SPLINE
SPL {X  -162.820, Y  +509.871, Z    +0.000, E1   +42.115, E3 +330842.346}
SPL {X  -162.820, Y  +501.934, Z    +0.000, E1   +43.022, E3 +330855.073}
SPL {X  -162.820, Y  +494.356, Z    +0.000, E1   +43.819, E3 +330866.915}
SPL {X  -162.820, Y  +487.058, Z    +0.000, E1   +44.544, E3 +330878.378}
SPL {X  -162.820, Y  +476.193, Z    +0.000, E1   +45.591, E3 +330894.817}
SPL {X  -162.820, Y  +465.836, Z    +0.000, E1   +46.727, E3 +330908.733}
SPL {X  -162.820, Y  +457.217, Z    +0.000, E1   +47.671, E3 +330919.772}
SPL {X  -162.820, Y  +446.677, Z    +0.000, E1   +48.707, E3 +330933.301}
SPL {X  -162.820, Y  +435.978, Z    +0.000, E1   +49.560, E3 +330947.450}
SPL {X  -162.820, Y  +428.488, Z    +0.000, E1   +49.830, E3 +330959.030}
SPL {X  -162.820, Y  +423.062, Z    +0.000, E1   +49.728, E3 +330969.173}
SPL {X  -162.820, Y  +416.560, Z    +0.000, E1   +49.816, E3 +330980.154}
SPL {X  -162.820, Y  +407.996, Z    +0.000, E1   +49.793, E3 +330995.519}
SPL {X  -162.820, Y  +398.766, Z    +0.000, E1   +49.793, E3 +331011.698}
SPL {X  -162.820, Y  +391.831, Z    +0.000, E1   +49.801, E3 +331023.744}
SPL {X  -162.820, Y  +386.334, Z    +0.000, E1   +49.739, E3 +331033.833}
SPL {X  -162.801, Y  +377.981, Z    +0.000, E1   +49.798, E3 +331048.354}
SPL {X  -162.314, Y  +367.677, Z    +0.000, E1   +49.734, E3 +331066.994}
SPL {X  -161.614, Y  +360.718, Z    +0.000, E1   +49.491, E3 +331080.412}
SPL {X  -160.828, Y  +355.106, Z    +0.000, E1   +49.536, E3 +331090.096}
SPL {X  -159.832, Y  +349.452, Z    +0.000, E1   +49.188, E3 +331102.067}
SPL {X  -158.863, Y  +344.823, Z    +0.000, E1   +49.020, E3 +331111.116}
SPL {X  -157.695, Y  +339.971, Z    +0.000, E1   +48.934, E3 +331120.212}
SPL {X  -156.136, Y  +334.326, Z    +0.000, E1   +48.578, E3 +331132.179}
SPL {X  -154.561, Y  +329.302, Z    +0.000, E1   +48.290, E3 +331142.509}
SPL {X  -152.787, Y  +324.229, Z    +0.000, E1   +47.981, E3 +331153.200}
SPL {X  -150.789, Y  +319.074, Z    +0.000, E1   +47.585, E3 +331164.222}
SPL {X  -145.123, Y  +306.679, Z    +0.000, E1   +50.518, E3 +331170.119}
SPL {X  -135.207, Y  +289.783, Z    +0.000, E1   +44.101, E3 +331263.634}
ENDSPLINE

SPLINE
SPL {X  -154.528, Y  +329.203, Z    +0.000, E1   +28.834, E3 +331333.995}
SPL {X  -160.380, Y  +352.419, Z    +0.000, E1   +18.163, E3 +331338.355}
SPL {X  -162.149, Y  +365.734, Z    +0.000, E1   +11.090, E3 +331336.964}
SPL {X  -162.754, Y  +375.862, Z    +0.000, E1    +5.134, E3 +331337.801}
SPL {X  -162.820, Y  +382.085, Z    +0.000, E1    +0.928, E3 +331337.489}
SPL {X  -162.820, Y  +385.149, Z    +0.000, E1    -1.602, E3 +331337.216}
SPL {X  -162.820, Y  +388.871, Z    +0.000, E1    -5.151, E3 +331337.171}
SPL {X  -162.820, Y  +395.861, Z    +0.000, E1   -13.028, E3 +331337.282}
SPL {X  -162.820, Y  +409.049, Z    +0.000, E1   -29.128, E3 +331336.125}
SPL {X  -162.820, Y  +446.299, Z    +0.000, E1   -49.360, E3 +331356.629}
SPL {X  -162.820, Y  +502.427, Z    +0.000, E1   -53.345, E3 +331419.614}
ENDSPLINE

SPLINE
SPL {X  -162.820, Y  +494.458, Z    +0.000, E1   -49.332, E3 +331430.146}
ENDSPLINE

SPLINE
SPL {X  -162.820, Y  +499.429, Z    +0.000, E1   -49.453, E3 +331438.355}
SPL {X  -162.820, Y  +505.173, Z    +0.000, E1   -49.386, E3 +331449.011}
SPL {X  -162.820, Y  +510.642, Z    +0.000, E1   -49.447, E3 +331458.361}
SPL {X  -162.820, Y  +516.435, Z    +0.000, E1   -49.526, E3 +331468.239}
SPL {X  -162.820, Y  +523.383, Z    +0.000, E1   -49.407, E3 +331481.426}
SPL {X  -162.820, Y  +530.598, Z    +0.000, E1   -49.471, E3 +331493.828}
SPL {X  -162.820, Y  +536.932, Z    +0.000, E1   -49.395, E3 +331505.585}
SPL {X  -162.820, Y  +543.021, Z    +0.000, E1   -49.432, E3 +331516.191}
SPL {X  -162.820, Y  +548.933, Z    +0.000, E1   -49.456, E3 +331526.595}
SPL {X  -162.820, Y  +553.997, Z    +0.000, E1   -49.325, E3 +331536.399}
SPL {X  -162.820, Y  +560.268, Z    +0.000, E1   -49.531, E3 +331546.357}
SPL {X  -162.820, Y  +564.590, Z    +0.000, E1   -49.361, E3 +331555.056}
SPL {X  -162.820, Y  +570.444, Z    +0.000, E1   -49.421, E3 +331565.208}
SPL {X  -162.820, Y  +577.429, Z    +0.000, E1   -49.474, E3 +331577.322}
SPL {X  -162.820, Y  +585.965, Z    +0.000, E1   -49.447, E3 +331592.896}
SPL {X  -162.820, Y  +594.192, Z    +0.000, E1   -49.325, E3 +331608.139}
SPL {X  -162.820, Y  +600.267, Z    +0.000, E1   -49.443, E3 +331618.228}
SPL {X  -162.820, Y  +606.218, Z    +0.000, E1   -49.464, E3 +331628.775}
SPL {X  -162.820, Y  +612.538, Z    +0.000, E1   -49.488, E3 +331639.826}
SPL {X  -162.820, Y  +617.738, Z    +0.000, E1   -49.301, E3 +331650.262}
SPL {X  -162.820, Y  +624.265, Z    +0.000, E1   -49.443, E3 +331661.057}
SPL {X  -162.820, Y  +632.551, Z    +0.000, E1   -49.478, E3 +331675.826}
SPL {X  -162.820, Y  +641.207, Z    +0.000, E1   -49.420, E3 +331691.469}
SPL {X  -162.820, Y  +649.864, Z    +0.000, E1   -49.433, E3 +331706.947}
SPL {X  -162.820, Y  +658.147, Z    +0.000, E1   -49.491, E3 +331721.214}
SPL {X  -162.820, Y  +663.916, Z    +0.000, E1   -49.371, E3 +331732.204}
SPL {X  -162.820, Y  +669.755, Z    +0.000, E1   -49.387, E3 +331742.529}
SPL {X  -162.807, Y  +675.597, Z    +0.000, E1   -49.472, E3 +331752.431}
SPL {X  -162.632, Y  +681.322, Z    +0.000, E1   -49.345, E3 +331763.443}
SPL {X  -162.228, Y  +687.372, Z    +0.000, E1   -49.294, E3 +331774.529}
SPL {X  -161.723, Y  +692.372, Z    +0.000, E1   -49.172, E3 +331784.159}
SPL {X  -161.009, Y  +697.714, Z    +0.000, E1   -49.214, E3 +331793.444}
SPL {X  -160.313, Y  +701.965, Z    +0.000, E1   -48.932, E3 +331802.656}
SPL {X  -158.980, Y  +708.651, Z    +0.000, E1   -48.774, E3 +331815.696}
SPL {X  -157.477, Y  +714.869, Z    +0.000, E1   -48.424, E3 +331828.571}
SPL {X  -156.071, Y  +719.891, Z    +0.000, E1   -48.264, E3 +331838.447}
SPL {X  -154.661, Y  +724.395, Z    +0.000, E1   -47.951, E3 +331848.129}
SPL {X  -153.094, Y  +728.931, Z    +0.000, E1   -47.705, E3 +331857.565}
SPL {X  -150.266, Y  +736.194, Z    +0.000, E1   -47.943, E3 +331869.174}
SPL {X  -143.458, Y  +750.508, Z    +0.000, E1   -51.034, E3 +331877.200}
SPL {X  -135.559, Y  +763.690, Z    +0.000, E1   -44.340, E3 +331961.445}
ENDSPLINE

SPLINE
SPL {X  -153.801, Y  +726.938, Z    +0.000, E1   -29.643, E3 +332030.158}
SPL {X  -160.383, Y  +701.564, Z    +0.000, E1   -18.145, E3 +332038.297}
SPL {X  -162.078, Y  +689.023, Z    +0.000, E1   -11.510, E3 +332037.835}
SPL {X  -162.685, Y  +680.136, Z    +0.000, E1    -6.379, E3 +332038.124}
SPL {X  -162.820, Y  +672.919, Z    +0.000, E1    -1.752, E3 +332038.163}
SPL {X  -162.820, Y  +667.861, Z    +0.000, E1    +2.254, E3 +332037.964}
SPL {X  -162.820, Y  +662.755, Z    +0.000, E1    +7.521, E3 +332038.005}
SPL {X  -162.820, Y  +657.537, Z    +0.000, E1   +13.540, E3 +332037.674}
SPL {X  -162.820, Y  +650.460, Z    +0.000, E1   +22.200, E3 +332037.105}
SPL {X  -162.820, Y  +637.843, Z    +0.000, E1   +35.051, E3 +332039.182}
SPL {X  -162.820, Y  +595.072, Z    +0.000, E1   +53.652, E3 +332059.902}
SPL {X  -162.820, Y  +561.831, Z    +0.000, E1   +49.171, E3 +332127.125}
SPL {X  -162.820, Y  +553.813, Z    +0.000, E1   +48.452, E3 +332146.190}
SPL {X  -162.820, Y  +543.226, Z    +0.000, E1   +48.398, E3 +332166.042}
SPL {X  -162.820, Y  +534.689, Z    +0.000, E1   +48.295, E3 +332182.343}
SPL {X  -162.820, Y  +528.564, Z    +0.000, E1   +48.407, E3 +332192.916}
SPL {X  -162.820, Y  +522.157, Z    +0.000, E1   +48.326, E3 +332205.497}
SPL {X  -162.820, Y  +513.750, Z    +0.000, E1   +48.520, E3 +332219.729}
SPL {X  -162.820, Y  +508.282, Z    +0.000, E1   +48.307, E3 +332231.131}
SPL {X  -162.820, Y  +502.890, Z    +0.000, E1   +48.309, E3 +332241.058}
ENDSPLINE

SPLINE
SPL {X  -162.820, Y  +520.386, Z    +0.000, E1   +40.911, E3 +332247.788}
ENDSPLINE

SPLINE
SPL {X  -162.820, Y  +515.876, Z    +0.000, E1   +41.348, E3 +332255.986}
SPL {X  -162.820, Y  +507.007, Z    +0.000, E1   +42.470, E3 +332270.000}
SPL {X  -162.820, Y  +496.780, Z    +0.000, E1   +43.573, E3 +332286.255}
SPL {X  -162.820, Y  +488.962, Z    +0.000, E1   +44.342, E3 +332298.523}
SPL {X  -162.820, Y  +481.373, Z    +0.000, E1   +45.107, E3 +332310.007}
SPL {X  -162.820, Y  +473.909, Z    +0.000, E1   +45.743, E3 +332321.520}
SPL {X  -162.820, Y  +463.464, Z    +0.000, E1   +47.025, E3 +332334.737}
SPL {X  -162.820, Y  +451.336, Z    +0.000, E1   +48.248, E3 +332350.507}
SPL {X  -162.820, Y  +443.046, Z    +0.000, E1   +49.021, E3 +332361.006}
SPL {X  -162.820, Y  +435.978, Z    +0.000, E1   +49.560, E3 +332370.527}
SPL {X  -162.820, Y  +428.488, Z    +0.000, E1   +49.830, E3 +332382.107}
SPL {X  -162.820, Y  +423.062, Z    +0.000, E1   +49.728, E3 +332392.250}
SPL {X  -162.820, Y  +416.560, Z    +0.000, E1   +49.816, E3 +332403.231}
SPL {X  -162.820, Y  +407.996, Z    +0.000, E1   +49.793, E3 +332418.596}
SPL {X  -162.820, Y  +400.367, Z    +0.000, E1   +49.822, E3 +332431.654}
SPL {X  -162.820, Y  +393.582, Z    +0.000, E1   +49.779, E3 +332443.972}
SPL {X  -162.820, Y  +384.205, Z    +0.000, E1   +49.756, E3 +332460.753}
SPL {X  -162.753, Y  +375.844, Z    +0.000, E1   +49.816, E3 +332474.928}
SPL {X  -162.415, Y  +369.029, Z    +0.000, E1   +49.751, E3 +332487.418}
SPL {X  -161.760, Y  +361.947, Z    +0.000, E1   +49.515, E3 +332501.256}
SPL {X  -160.828, Y  +355.106, Z    +0.000, E1   +49.536, E3 +332513.173}
SPL {X  -159.832, Y  +349.452, Z    +0.000, E1   +49.188, E3 +332525.144}
SPL {X  -158.863, Y  +344.823, Z    +0.000, E1   +49.020, E3 +332534.193}
SPL {X  -157.695, Y  +339.971, Z    +0.000, E1   +48.934, E3 +332543.289}
SPL {X  -156.136, Y  +334.326, Z    +0.000, E1   +48.578, E3 +332555.256}
SPL {X  -154.561, Y  +329.302, Z    +0.000, E1   +48.290, E3 +332565.586}
SPL {X  -152.787, Y  +324.229, Z    +0.000, E1   +47.981, E3 +332576.276}
SPL {X  -150.789, Y  +319.074, Z    +0.000, E1   +47.585, E3 +332587.299}
SPL {X  -145.123, Y  +306.679, Z    +0.000, E1   +50.518, E3 +332593.196}
SPL {X  -135.207, Y  +289.783, Z    +0.000, E1   +44.101, E3 +332686.711}
ENDSPLINE

SPLINE
SPL {X  -154.528, Y  +329.203, Z    +0.000, E1   +28.834, E3 +332757.072}
SPL {X  -160.380, Y  +352.419, Z    +0.000, E1   +18.163, E3 +332761.432}
SPL {X  -162.408, Y  +368.921, Z    +0.000, E1    +9.337, E3 +332760.182}
SPL {X  -162.817, Y  +379.558, Z    +0.000, E1    +2.744, E3 +332760.572}
SPL {X  -162.820, Y  +383.077, Z    +0.000, E1    +0.110, E3 +332760.968}
SPL {X  -162.820, Y  +386.028, Z    +0.000, E1    -2.328, E3 +332760.291}
SPL {X  -162.820, Y  +389.792, Z    +0.000, E1    -6.211, E3 +332760.223}
SPL {X  -162.820, Y  +395.861, Z    +0.000, E1   -13.028, E3 +332760.359}
SPL {X  -162.820, Y  +409.049, Z    +0.000, E1   -29.128, E3 +332759.202}
SPL {X  -162.820, Y  +446.299, Z    +0.000, E1   -49.360, E3 +332779.705}
SPL {X  -162.820, Y  +502.427, Z    +0.000, E1   -53.345, E3 +332842.691}
ENDSPLINE

SPLINE
SPL {X  -162.820, Y  +494.458, Z    +0.000, E1   -49.332, E3 +332853.223}
ENDSPLINE

SPLINE
SPL {X  -162.820, Y  +499.429, Z    +0.000, E1   -49.453, E3 +332861.432}
SPL {X  -162.820, Y  +505.173, Z    +0.000, E1   -49.386, E3 +332872.088}
SPL {X  -162.820, Y  +510.642, Z    +0.000, E1   -49.447, E3 +332881.438}
SPL {X  -162.820, Y  +516.435, Z    +0.000, E1   -49.526, E3 +332891.316}
SPL {X  -162.820, Y  +522.095, Z    +0.000, E1   -49.420, E3 +332902.013}
SPL {X  -162.820, Y  +529.397, Z    +0.000, E1   -49.440, E3 +332915.021}
SPL {X  -162.820, Y  +536.932, Z    +0.000, E1   -49.395, E3 +332928.662}
SPL {X  -162.820, Y  +543.021, Z    +0.000, E1   -49.432, E3 +332939.268}
SPL {X  -162.820, Y  +548.933, Z    +0.000, E1   -49.456, E3 +332949.672}
SPL {X  -162.820, Y  +553.997, Z    +0.000, E1   -49.325, E3 +332959.476}
SPL {X  -162.820, Y  +562.346, Z    +0.000, E1   -49.498, E3 +332973.538}
SPL {X  -162.820, Y  +570.444, Z    +0.000, E1   -49.421, E3 +332988.285}
SPL {X  -162.820, Y  +577.429, Z    +0.000, E1   -49.474, E3 +333000.399}
SPL {X  -162.820, Y  +585.965, Z    +0.000, E1   -49.447, E3 +333015.973}
SPL {X  -162.820, Y  +594.192, Z    +0.000, E1   -49.325, E3 +333031.216}
SPL {X  -162.820, Y  +600.267, Z    +0.000, E1   -49.443, E3 +333041.305}
SPL {X  -162.820, Y  +606.218, Z    +0.000, E1   -49.464, E3 +333051.851}
SPL {X  -162.820, Y  +612.538, Z    +0.000, E1   -49.488, E3 +333062.902}
SPL {X  -162.820, Y  +617.738, Z    +0.000, E1   -49.301, E3 +333073.339}
SPL {X  -162.820, Y  +624.265, Z    +0.000, E1   -49.443, E3 +333084.134}
SPL {X  -162.820, Y  +632.551, Z    +0.000, E1   -49.478, E3 +333098.903}
SPL {X  -162.820, Y  +641.207, Z    +0.000, E1   -49.420, E3 +333114.546}
SPL {X  -162.820, Y  +649.864, Z    +0.000, E1   -49.433, E3 +333130.024}
SPL {X  -162.820, Y  +658.147, Z    +0.000, E1   -49.491, E3 +333144.291}
SPL {X  -162.820, Y  +663.916, Z    +0.000, E1   -49.371, E3 +333155.281}
SPL {X  -162.820, Y  +669.755, Z    +0.000, E1   -49.387, E3 +333165.606}
SPL {X  -162.807, Y  +675.597, Z    +0.000, E1   -49.472, E3 +333175.508}
SPL {X  -162.632, Y  +681.322, Z    +0.000, E1   -49.345, E3 +333186.520}
SPL {X  -162.228, Y  +687.372, Z    +0.000, E1   -49.294, E3 +333197.606}
SPL {X  -161.723, Y  +692.372, Z    +0.000, E1   -49.172, E3 +333207.236}
SPL {X  -161.009, Y  +697.714, Z    +0.000, E1   -49.214, E3 +333216.521}
SPL {X  -160.313, Y  +701.965, Z    +0.000, E1   -48.932, E3 +333225.733}
SPL {X  -158.980, Y  +708.651, Z    +0.000, E1   -48.774, E3 +333238.773}
SPL {X  -157.477, Y  +714.869, Z    +0.000, E1   -48.424, E3 +333251.648}
SPL {X  -156.071, Y  +719.891, Z    +0.000, E1   -48.264, E3 +333261.524}
SPL {X  -154.661, Y  +724.395, Z    +0.000, E1   -47.951, E3 +333271.206}
SPL {X  -153.094, Y  +728.931, Z    +0.000, E1   -47.705, E3 +333280.642}
SPL {X  -151.300, Y  +733.655, Z    +0.000, E1   -47.339, E3 +333290.951}
SPL {X  -145.669, Y  +746.239, Z    +0.000, E1   -50.198, E3 +333297.727}
SPL {X  -135.084, Y  +764.399, Z    +0.000, E1   -44.787, E3 +333380.631}
ENDSPLINE

SPLINE
SPL {X  -153.038, Y  +729.086, Z    +0.000, E1   -30.522, E3 +333451.338}
SPL {X  -160.383, Y  +701.564, Z    +0.000, E1   -18.145, E3 +333461.374}
SPL {X  -162.078, Y  +689.023, Z    +0.000, E1   -11.510, E3 +333460.912}
SPL {X  -162.685, Y  +680.136, Z    +0.000, E1    -6.379, E3 +333461.201}
SPL {X  -162.820, Y  +672.919, Z    +0.000, E1    -1.752, E3 +333461.240}
SPL {X  -162.820, Y  +667.861, Z    +0.000, E1    +2.254, E3 +333461.041}
SPL {X  -162.820, Y  +662.755, Z    +0.000, E1    +7.521, E3 +333461.082}
SPL {X  -162.820, Y  +657.537, Z    +0.000, E1   +13.540, E3 +333460.751}
SPL {X  -162.820, Y  +650.460, Z    +0.000, E1   +22.200, E3 +333460.182}
SPL {X  -162.820, Y  +641.200, Z    +0.000, E1   +31.596, E3 +333462.806}
SPL {X  -162.820, Y  +634.978, Z    +0.000, E1   +38.045, E3 +333461.791}
SPL {X  -162.820, Y  +595.072, Z    +0.000, E1   +53.652, E3 +333482.979}
SPL {X  -162.820, Y  +561.831, Z    +0.000, E1   +49.171, E3 +333550.201}
SPL {X  -162.820, Y  +555.289, Z    +0.000, E1   +48.406, E3 +333566.663}
SPL {X  -162.820, Y  +547.003, Z    +0.000, E1   +48.390, E3 +333582.075}
SPL {X  -162.820, Y  +540.645, Z    +0.000, E1   +48.364, E3 +333593.871}
SPL {X  -162.820, Y  +534.689, Z    +0.000, E1   +48.295, E3 +333605.420}
SPL {X  -162.820, Y  +526.053, Z    +0.000, E1   +48.382, E3 +333620.995}
SPL {X  -162.820, Y  +519.666, Z    +0.000, E1   +48.261, E3 +333633.364}
SPL {X  -162.820, Y  +513.750, Z    +0.000, E1   +48.520, E3 +333642.806}
SPL {X  -162.820, Y  +508.282, Z    +0.000, E1   +48.307, E3 +333654.208}
SPL {X  -162.820, Y  +502.890, Z    +0.000, E1   +48.309, E3 +333664.135}
ENDSPLINE

SPLINE
SPL {X  -162.820, Y  +517.326, Z    +0.000, E1   +41.232, E3 +333676.399}
ENDSPLINE

SPLINE
SPL {X  -162.820, Y  +509.871, Z    +0.000, E1   +42.115, E3 +333688.500}
SPL {X  -162.820, Y  +501.934, Z    +0.000, E1   +43.022, E3 +333701.227}
SPL {X  -162.820, Y  +494.356, Z    +0.000, E1   +43.819, E3 +333713.069}
SPL {X  -162.820, Y  +487.058, Z    +0.000, E1   +44.544, E3 +333724.532}
SPL {X  -162.820, Y  +476.193, Z    +0.000, E1   +45.591, E3 +333740.971}
SPL {X  -162.820, Y  +465.836, Z    +0.000, E1   +46.727, E3 +333754.887}
SPL {X  -162.820, Y  +457.217, Z    +0.000, E1   +47.671, E3 +333765.925}
SPL {X  -162.820, Y  +449.104, Z    +0.000, E1   +48.459, E3 +333776.394}
SPL {X  -162.820, Y  +438.072, Z    +0.000, E1   +49.432, E3 +333790.749}
SPL {X  -162.820, Y  +428.488, Z    +0.000, E1   +49.830, E3 +333805.184}
SPL {X  -162.820, Y  +423.062, Z    +0.000, E1   +49.728, E3 +333815.327}
SPL {X  -162.820, Y  +416.560, Z    +0.000, E1   +49.816, E3 +333826.307}
SPL {X  -162.820, Y  +410.559, Z    +0.000, E1   +49.727, E3 +333837.363}
SPL {X  -162.820, Y  +405.170, Z    +0.000, E1   +49.772, E3 +333846.565}
SPL {X  -162.820, Y  +398.766, Z    +0.000, E1   +49.793, E3 +333857.852}
SPL {X  -162.820, Y  +391.831, Z    +0.000, E1   +49.801, E3 +333869.898}
SPL {X  -162.820, Y  +386.334, Z    +0.000, E1   +49.739, E3 +333879.986}
SPL {X  -162.801, Y  +377.981, Z    +0.000, E1   +49.798, E3 +333894.508}
SPL {X  -162.314, Y  +367.677, Z    +0.000, E1   +49.734, E3 +333913.148}
SPL {X  -161.359, Y  +358.734, Z    +0.000, E1   +49.535, E3 +333929.932}
SPL {X  -160.051, Y  +350.597, Z    +0.000, E1   +49.332, E3 +333945.542}
SPL {X  -158.863, Y  +344.823, Z    +0.000, E1   +49.020, E3 +333957.270}
SPL {X  -157.695, Y  +339.971, Z    +0.000, E1   +48.934, E3 +333966.366}
SPL {X  -156.136, Y  +334.326, Z    +0.000, E1   +48.578, E3 +333978.332}
SPL {X  -154.561, Y  +329.302, Z    +0.000, E1   +48.290, E3 +333988.663}
SPL {X  -152.787, Y  +324.229, Z    +0.000, E1   +47.981, E3 +333999.353}
SPL {X  -150.789, Y  +319.074, Z    +0.000, E1   +47.585, E3 +334010.376}
SPL {X  -145.123, Y  +306.679, Z    +0.000, E1   +50.518, E3 +334016.273}
SPL {X  -135.207, Y  +289.783, Z    +0.000, E1   +44.101, E3 +334109.788}
ENDSPLINE

SPLINE
SPL {X  -154.528, Y  +329.203, Z    +0.000, E1   +28.834, E3 +334180.149}
SPL {X  -160.380, Y  +352.419, Z    +0.000, E1   +18.163, E3 +334184.509}
SPL {X  -162.149, Y  +365.734, Z    +0.000, E1   +11.090, E3 +334183.118}
SPL {X  -162.754, Y  +375.862, Z    +0.000, E1    +5.134, E3 +334183.955}
SPL {X  -162.820, Y  +382.085, Z    +0.000, E1    +0.928, E3 +334183.643}
SPL {X  -162.820, Y  +386.028, Z    +0.000, E1    -2.328, E3 +334183.368}
SPL {X  -162.820, Y  +389.792, Z    +0.000, E1    -6.211, E3 +334183.300}
SPL {X  -162.820, Y  +394.068, Z    +0.000, E1   -11.043, E3 +334183.417}
SPL {X  -162.820, Y  +398.921, Z    +0.000, E1   -16.945, E3 +334183.470}
SPL {X  -162.820, Y  +409.049, Z    +0.000, E1   -29.128, E3 +334182.279}
SPL {X  -162.820, Y  +446.299, Z    +0.000, E1   -49.360, E3 +334202.782}
SPL {X  -162.820, Y  +502.427, Z    +0.000, E1   -53.345, E3 +334265.768}
ENDSPLINE

SPLINE
SPL {X  -162.820, Y  +497.758, Z    +0.000, E1   -49.444, E3 +334281.707}
ENDSPLINE

SPLINE
SPL {X  -162.820, Y  +507.703, Z    +0.000, E1   -49.462, E3 +334299.424}
SPL {X  -162.820, Y  +516.435, Z    +0.000, E1   -49.526, E3 +334314.393}
SPL {X  -162.820, Y  +522.095, Z    +0.000, E1   -49.420, E3 +334325.090}
SPL {X  -162.820, Y  +529.397, Z    +0.000, E1   -49.440, E3 +334338.098}
SPL {X  -162.820, Y  +536.932, Z    +0.000, E1   -49.395, E3 +334351.739}
SPL {X  -162.820, Y  +543.021, Z    +0.000, E1   -49.432, E3 +334362.345}
SPL {X  -162.820, Y  +548.933, Z    +0.000, E1   -49.456, E3 +334372.749}
SPL {X  -162.820, Y  +553.997, Z    +0.000, E1   -49.325, E3 +334382.553}
SPL {X  -162.820, Y  +562.346, Z    +0.000, E1   -49.498, E3 +334396.615}
SPL {X  -162.820, Y  +570.444, Z    +0.000, E1   -49.421, E3 +334411.362}
SPL {X  -162.820, Y  +577.429, Z    +0.000, E1   -49.474, E3 +334423.476}
SPL {X  -162.820, Y  +582.387, Z    +0.000, E1   -49.269, E3 +334433.497}
SPL {X  -162.820, Y  +588.456, Z    +0.000, E1   -49.496, E3 +334443.012}
SPL {X  -162.820, Y  +594.192, Z    +0.000, E1   -49.325, E3 +334454.293}
SPL {X  -162.820, Y  +600.267, Z    +0.000, E1   -49.443, E3 +334464.382}
SPL {X  -162.820, Y  +606.218, Z    +0.000, E1   -49.464, E3 +334474.928}
SPL {X  -162.820, Y  +612.538, Z    +0.000, E1   -49.488, E3 +334485.979}
SPL {X  -162.820, Y  +617.738, Z    +0.000, E1   -49.301, E3 +334496.416}
SPL {X  -162.820, Y  +624.265, Z    +0.000, E1   -49.443, E3 +334507.211}
SPL {X  -162.820, Y  +632.551, Z    +0.000, E1   -49.478, E3 +334521.980}
SPL {X  -162.820, Y  +641.207, Z    +0.000, E1   -49.420, E3 +334537.623}
SPL {X  -162.820, Y  +648.011, Z    +0.000, E1   -49.484, E3 +334549.300}
SPL {X  -162.820, Y  +655.976, Z    +0.000, E1   -49.445, E3 +334563.929}
SPL {X  -162.820, Y  +663.916, Z    +0.000, E1   -49.371, E3 +334578.358}
SPL {X  -162.820, Y  +669.755, Z    +0.000, E1   -49.387, E3 +334588.683}
SPL {X  -162.807, Y  +675.597, Z    +0.000, E1   -49.472, E3 +334598.585}
SPL {X  -162.632, Y  +681.322, Z    +0.000, E1   -49.345, E3 +334609.596}
SPL {X  -162.228, Y  +687.372, Z    +0.000, E1   -49.294, E3 +334620.683}
SPL {X  -161.723, Y  +692.372, Z    +0.000, E1   -49.172, E3 +334630.313}
SPL {X  -161.009, Y  +697.714, Z    +0.000, E1   -49.214, E3 +334639.598}
SPL {X  -160.313, Y  +701.965, Z    +0.000, E1   -48.932, E3 +334648.810}
SPL {X  -159.435, Y  +706.528, Z    +0.000, E1   -48.764, E3 +334657.937}
SPL {X  -157.894, Y  +713.249, Z    +0.000, E1   -48.586, E3 +334671.130}
SPL {X  -156.071, Y  +719.891, Z    +0.000, E1   -48.264, E3 +334684.601}
SPL {X  -154.661, Y  +724.395, Z    +0.000, E1   -47.951, E3 +334694.282}
SPL {X  -153.094, Y  +728.931, Z    +0.000, E1   -47.705, E3 +334703.719}
SPL {X  -151.300, Y  +733.655, Z    +0.000, E1   -47.339, E3 +334714.028}
SPL {X  -145.669, Y  +746.239, Z    +0.000, E1   -50.198, E3 +334720.804}
SPL {X  -135.084, Y  +764.399, Z    +0.000, E1   -44.787, E3 +334803.708}
ENDSPLINE

SPLINE
SPL {X  -153.038, Y  +729.086, Z    +0.000, E1   -30.522, E3 +334874.415}
SPL {X  -160.383, Y  +701.564, Z    +0.000, E1   -18.145, E3 +334884.451}
SPL {X  -162.078, Y  +689.023, Z    +0.000, E1   -11.510, E3 +334883.989}
SPL {X  -162.685, Y  +680.136, Z    +0.000, E1    -6.379, E3 +334884.278}
SPL {X  -162.820, Y  +672.919, Z    +0.000, E1    -1.752, E3 +334884.317}
SPL {X  -162.820, Y  +669.270, Z    +0.000, E1    +1.140, E3 +334883.799}
SPL {X  -162.820, Y  +666.754, Z    +0.000, E1    +3.396, E3 +334884.368}
SPL {X  -162.820, Y  +662.755, Z    +0.000, E1    +7.521, E3 +334884.159}
SPL {X  -162.820, Y  +657.537, Z    +0.000, E1   +13.540, E3 +334883.828}
SPL {X  -162.820, Y  +650.460, Z    +0.000, E1   +22.200, E3 +334883.259}
SPL {X  -162.820, Y  +637.843, Z    +0.000, E1   +35.051, E3 +334885.336}
SPL {X  -162.820, Y  +595.072, Z    +0.000, E1   +53.652, E3 +334906.056}
SPL {X  -162.820, Y  +560.706, Z    +0.000, E1   +50.482, E3 +334966.965}
ENDSPLINE

SPLINE
SPL {X  -162.820, Y  +560.978, Z    +0.000, E1   +48.448, E3 +334979.051}
ENDSPLINE

SPLINE
SPL {X  -162.820, Y  +552.125, Z    +0.000, E1   +48.477, E3 +334995.155}
SPL {X  -162.820, Y  +545.800, Z    +0.000, E1   +48.334, E3 +335007.597}
SPL {X  -162.820, Y  +540.645, Z    +0.000, E1   +48.364, E3 +335016.948}
SPL {X  -162.820, Y  +534.689, Z    +0.000, E1   +48.295, E3 +335028.497}
SPL {X  -162.820, Y  +526.053, Z    +0.000, E1   +48.382, E3 +335044.072}
SPL {X  -162.820, Y  +519.666, Z    +0.000, E1   +48.261, E3 +335056.440}
SPL {X  -162.820, Y  +512.600, Z    +0.000, E1   +48.469, E3 +335068.427}
SPL {X  -162.820, Y  +504.728, Z    +0.000, E1   +48.342, E3 +335083.756}
ENDSPLINE

SPLINE
SPL {X  -162.820, Y  +517.326, Z    +0.000, E1   +41.232, E3 +335099.476}
ENDSPLINE

SPLINE
SPL {X  -162.820, Y  +509.871, Z    +0.000, E1   +42.115, E3 +335111.577}
SPL {X  -162.820, Y  +501.934, Z    +0.000, E1   +43.022, E3 +335124.304}
SPL {X  -162.820, Y  +494.356, Z    +0.000, E1   +43.819, E3 +335136.145}
SPL {X  -162.820, Y  +487.058, Z    +0.000, E1   +44.544, E3 +335147.609}
SPL {X  -162.820, Y  +476.193, Z    +0.000, E1   +45.591, E3 +335164.048}
SPL {X  -162.820, Y  +465.836, Z    +0.000, E1   +46.727, E3 +335177.964}
SPL {X  -162.820, Y  +457.217, Z    +0.000, E1   +47.671, E3 +335189.002}
SPL {X  -162.820, Y  +446.677, Z    +0.000, E1   +48.707, E3 +335202.532}
SPL {X  -162.820, Y  +435.978, Z    +0.000, E1   +49.560, E3 +335216.681}
SPL {X  -162.820, Y  +428.488, Z    +0.000, E1   +49.830, E3 +335228.261}
SPL {X  -162.820, Y  +423.062, Z    +0.000, E1   +49.728, E3 +335238.403}
SPL {X  -162.820, Y  +416.560, Z    +0.000, E1   +49.816, E3 +335249.384}
SPL {X  -162.820, Y  +407.996, Z    +0.000, E1   +49.793, E3 +335264.750}
SPL {X  -162.820, Y  +398.766, Z    +0.000, E1   +49.793, E3 +335280.929}
SPL {X  -162.820, Y  +391.831, Z    +0.000, E1   +49.801, E3 +335292.975}
SPL {X  -162.820, Y  +386.334, Z    +0.000, E1   +49.739, E3 +335303.063}
SPL {X  -162.801, Y  +377.981, Z    +0.000, E1   +49.798, E3 +335317.585}
SPL {X  -162.314, Y  +367.677, Z    +0.000, E1   +49.734, E3 +335336.225}
SPL {X  -161.359, Y  +358.734, Z    +0.000, E1   +49.535, E3 +335353.008}
SPL {X  -160.051, Y  +350.597, Z    +0.000, E1   +49.332, E3 +335368.619}
SPL {X  -158.863, Y  +344.823, Z    +0.000, E1   +49.020, E3 +335380.347}
SPL {X  -157.695, Y  +339.971, Z    +0.000, E1   +48.934, E3 +335389.443}
SPL {X  -156.136, Y  +334.326, Z    +0.000, E1   +48.578, E3 +335401.409}
SPL {X  -153.956, Y  +327.511, Z    +0.000, E1   +48.205, E3 +335415.531}
SPL {X  -151.655, Y  +321.245, Z    +0.000, E1   +47.770, E3 +335428.741}
SPL {X  -148.347, Y  +313.391, Z    +0.000, E1   +48.924, E3 +335436.338}
SPL {X  -143.047, Y  +302.732, Z    +0.000, E1   +51.043, E3 +335442.858}
SPL {X  -135.207, Y  +289.783, Z    +0.000, E1   +44.101, E3 +335532.865}
ENDSPLINE

SPLINE
SPL {X  -154.528, Y  +329.203, Z    +0.000, E1   +28.834, E3 +335603.226}
SPL {X  -160.380, Y  +352.419, Z    +0.000, E1   +18.163, E3 +335607.586}
SPL {X  -162.149, Y  +365.734, Z    +0.000, E1   +11.090, E3 +335606.195}
SPL {X  -162.754, Y  +375.862, Z    +0.000, E1    +5.134, E3 +335607.031}
SPL {X  -162.820, Y  +382.085, Z    +0.000, E1    +0.928, E3 +335606.720}
SPL {X  -162.820, Y  +385.149, Z    +0.000, E1    -1.602, E3 +335606.447}
SPL {X  -162.820, Y  +388.871, Z    +0.000, E1    -5.151, E3 +335606.402}
SPL {X  -162.820, Y  +395.861, Z    +0.000, E1   -13.028, E3 +335606.513}
SPL {X  -162.820, Y  +409.049, Z    +0.000, E1   -29.128, E3 +335605.356}
SPL {X  -162.820, Y  +444.592, Z    +0.000, E1   -49.032, E3 +335624.365}
SPL {X  -162.820, Y  +458.217, Z    +0.000, E1   -51.268, E3 +335636.311}
SPL {X  -162.820, Y  +501.848, Z    +0.000, E1   -54.235, E3 +335682.679}
ENDSPLINE

SPLINE
SPL {X  -162.820, Y  +498.156, Z    +0.000, E1   -50.986, E3 +335696.228}
ENDSPLINE

SPLINE
SPL {X  -162.820, Y  +499.429, Z    +0.000, E1   -49.453, E3 +335707.586}
SPL {X  -162.820, Y  +507.703, Z    +0.000, E1   -49.462, E3 +335722.501}
SPL {X  -162.820, Y  +516.435, Z    +0.000, E1   -49.526, E3 +335737.470}
SPL {X  -162.820, Y  +523.383, Z    +0.000, E1   -49.407, E3 +335750.657}
SPL {X  -162.820, Y  +532.283, Z    +0.000, E1   -49.462, E3 +335766.259}
SPL {X  -162.820, Y  +541.471, Z    +0.000, E1   -49.456, E3 +335782.637}
SPL {X  -162.820, Y  +548.933, Z    +0.000, E1   -49.456, E3 +335795.826}
SPL {X  -162.820, Y  +553.997, Z    +0.000, E1   -49.325, E3 +335805.630}
SPL {X  -162.820, Y  +560.268, Z    +0.000, E1   -49.531, E3 +335815.587}
SPL {X  -162.820, Y  +564.590, Z    +0.000, E1   -49.361, E3 +335824.287}
SPL {X  -162.820, Y  +570.444, Z    +0.000, E1   -49.421, E3 +335834.439}
SPL {X  -162.820, Y  +577.429, Z    +0.000, E1   -49.474, E3 +335846.553}
SPL {X  -162.820, Y  +585.965, Z    +0.000, E1   -49.447, E3 +335862.127}
SPL {X  -162.820, Y  +594.192, Z    +0.000, E1   -49.325, E3 +335877.370}
SPL {X  -162.820, Y  +600.267, Z    +0.000, E1   -49.443, E3 +335887.458}
SPL {X  -162.820, Y  +606.218, Z    +0.000, E1   -49.464, E3 +335898.005}
SPL {X  -162.820, Y  +612.538, Z    +0.000, E1   -49.488, E3 +335909.056}
SPL {X  -162.820, Y  +617.738, Z    +0.000, E1   -49.301, E3 +335919.493}
SPL {X  -162.820, Y  +624.265, Z    +0.000, E1   -49.443, E3 +335930.288}
SPL {X  -162.820, Y  +632.551, Z    +0.000, E1   -49.478, E3 +335945.057}
SPL {X  -162.820, Y  +641.207, Z    +0.000, E1   -49.420, E3 +335960.700}
SPL {X  -162.820, Y  +649.864, Z    +0.000, E1   -49.433, E3 +335976.178}
SPL {X  -162.820, Y  +658.147, Z    +0.000, E1   -49.491, E3 +335990.445}
SPL {X  -162.820, Y  +663.916, Z    +0.000, E1   -49.371, E3 +336001.435}
SPL {X  -162.820, Y  +669.755, Z    +0.000, E1   -49.387, E3 +336011.760}
SPL {X  -162.807, Y  +675.597, Z    +0.000, E1   -49.472, E3 +336021.662}
SPL {X  -162.632, Y  +681.322, Z    +0.000, E1   -49.345, E3 +336032.673}
SPL {X  -162.228, Y  +687.372, Z    +0.000, E1   -49.294, E3 +336043.760}
SPL {X  -161.723, Y  +692.372, Z    +0.000, E1   -49.172, E3 +336053.390}
SPL {X  -161.009, Y  +697.714, Z    +0.000, E1   -49.214, E3 +336062.675}
SPL {X  -160.313, Y  +701.965, Z    +0.000, E1   -48.932, E3 +336071.887}
SPL {X  -158.980, Y  +708.651, Z    +0.000, E1   -48.774, E3 +336084.927}
SPL {X  -157.477, Y  +714.869, Z    +0.000, E1   -48.424, E3 +336097.802}
SPL {X  -156.071, Y  +719.891, Z    +0.000, E1   -48.264, E3 +336107.678}
SPL {X  -154.661, Y  +724.395, Z    +0.000, E1   -47.951, E3 +336117.359}
SPL {X  -153.094, Y  +728.931, Z    +0.000, E1   -47.705, E3 +336126.796}
SPL {X  -151.300, Y  +733.655, Z    +0.000, E1   -47.339, E3 +336137.105}
SPL {X  -145.669, Y  +746.239, Z    +0.000, E1   -50.198, E3 +336143.881}
SPL {X  -135.084, Y  +764.399, Z    +0.000, E1   -44.787, E3 +336226.785}
ENDSPLINE

SPLINE
SPL {X  -153.038, Y  +729.086, Z    +0.000, E1   -30.522, E3 +336297.492}
SPL {X  -160.383, Y  +701.564, Z    +0.000, E1   -18.145, E3 +336307.528}
SPL {X  -162.078, Y  +689.023, Z    +0.000, E1   -11.510, E3 +336307.066}
SPL {X  -162.685, Y  +680.136, Z    +0.000, E1    -6.379, E3 +336307.355}
SPL {X  -162.820, Y  +672.919, Z    +0.000, E1    -1.752, E3 +336307.394}
SPL {X  -162.820, Y  +669.270, Z    +0.000, E1    +1.140, E3 +336306.876}
SPL {X  -162.820, Y  +666.754, Z    +0.000, E1    +3.396, E3 +336307.445}
SPL {X  -162.820, Y  +662.755, Z    +0.000, E1    +7.521, E3 +336307.235}
SPL {X  -162.820, Y  +657.537, Z    +0.000, E1   +13.540, E3 +336306.905}
SPL {X  -162.820, Y  +650.460, Z    +0.000, E1   +22.200, E3 +336306.336}
SPL {X  -162.820, Y  +637.843, Z    +0.000, E1   +35.051, E3 +336308.413}
SPL {X  -162.820, Y  +595.072, Z    +0.000, E1   +53.652, E3 +336329.133}
SPL {X  -162.820, Y  +560.706, Z    +0.000, E1   +50.482, E3 +336390.042}
ENDSPLINE

SPLINE
SPL {X  -162.820, Y  +560.978, Z    +0.000, E1   +48.448, E3 +336402.128}
ENDSPLINE

SPLINE
SPL {X  -162.820, Y  +552.125, Z    +0.000, E1   +48.477, E3 +336418.232}
SPL {X  -162.820, Y  +545.800, Z    +0.000, E1   +48.334, E3 +336430.674}
SPL {X  -162.820, Y  +538.900, Z    +0.000, E1   +48.334, E3 +336443.589}
SPL {X  -162.820, Y  +530.572, Z    +0.000, E1   +48.392, E3 +336458.639}
SPL {X  -162.820, Y  +524.414, Z    +0.000, E1   +48.297, E3 +336470.522}
SPL {X  -162.820, Y  +516.130, Z    +0.000, E1   +48.458, E3 +336485.107}
SPL {X  -162.820, Y  +508.282, Z    +0.000, E1   +48.307, E3 +336500.362}
SPL {X  -162.820, Y  +502.890, Z    +0.000, E1   +48.309, E3 +336510.289}
ENDSPLINE

SPLINE
SPL {X  -162.820, Y  +517.326, Z    +0.000, E1   +41.232, E3 +336522.553}
ENDSPLINE

SPLINE
SPL {X  -162.820, Y  +507.007, Z    +0.000, E1   +42.470, E3 +336539.231}
SPL {X  -162.820, Y  +496.780, Z    +0.000, E1   +43.573, E3 +336555.486}
SPL {X  -162.820, Y  +488.962, Z    +0.000, E1   +44.342, E3 +336567.753}
SPL {X  -162.820, Y  +481.373, Z    +0.000, E1   +45.107, E3 +336579.238}
SPL {X  -162.820, Y  +473.909, Z    +0.000, E1   +45.743, E3 +336590.750}
SPL {X  -162.820, Y  +465.836, Z    +0.000, E1   +46.727, E3 +336601.041}
SPL {X  -162.820, Y  +457.217, Z    +0.000, E1   +47.671, E3 +336612.079}
SPL {X  -162.820, Y  +449.104, Z    +0.000, E1   +48.459, E3 +336622.548}
SPL {X  -162.820, Y  +440.303, Z    +0.000, E1   +49.204, E3 +336634.185}
SPL {X  -162.820, Y  +430.072, Z    +0.000, E1   +49.865, E3 +336648.487}
SPL {X  -162.820, Y  +423.062, Z    +0.000, E1   +49.728, E3 +336661.480}
SPL {X  -162.820, Y  +416.560, Z    +0.000, E1   +49.816, E3 +336672.461}
SPL {X  -162.820, Y  +410.559, Z    +0.000, E1   +49.727, E3 +336683.517}
SPL {X  -162.820, Y  +405.170, Z    +0.000, E1   +49.772, E3 +336692.719}
SPL {X  -162.820, Y  +398.766, Z    +0.000, E1   +49.793, E3 +336704.006}
SPL {X  -162.820, Y  +391.831, Z    +0.000, E1   +49.801, E3 +336716.052}
SPL {X  -162.820, Y  +386.334, Z    +0.000, E1   +49.739, E3 +336726.140}
SPL {X  -162.820, Y  +381.297, Z    +0.000, E1   +49.665, E3 +336735.411}
SPL {X  -162.709, Y  +374.487, Z    +0.000, E1   +49.773, E3 +336746.936}
SPL {X  -162.299, Y  +367.483, Z    +0.000, E1   +49.784, E3 +336759.078}
SPL {X  -161.760, Y  +361.947, Z    +0.000, E1   +49.515, E3 +336770.487}
SPL {X  -160.828, Y  +355.106, Z    +0.000, E1   +49.536, E3 +336782.403}
SPL {X  -159.832, Y  +349.452, Z    +0.000, E1   +49.188, E3 +336794.375}
SPL {X  -158.863, Y  +344.823, Z    +0.000, E1   +49.020, E3 +336803.424}
SPL {X  -157.695, Y  +339.971, Z    +0.000, E1   +48.934, E3 +336812.520}
SPL {X  -156.496, Y  +335.563, Z    +0.000, E1   +48.599, E3 +336822.097}
SPL {X  -154.894, Y  +330.318, Z    +0.000, E1   +48.380, E3 +336832.640}
SPL {X  -153.352, Y  +325.786, Z    +0.000, E1   +48.028, E3 +336842.397}
SPL {X  -151.316, Y  +320.384, Z    +0.000, E1   +47.734, E3 +336853.612}
SPL {X  -145.123, Y  +306.679, Z    +0.000, E1   +50.518, E3 +336862.427}
SPL {X  -135.207, Y  +289.783, Z    +0.000, E1   +44.101, E3 +336955.942}
ENDSPLINE

SPLINE
SPL {X  -154.528, Y  +329.203, Z    +0.000, E1   +28.834, E3 +337026.303}
SPL {X  -160.380, Y  +352.419, Z    +0.000, E1   +18.163, E3 +337030.663}
SPL {X  -162.408, Y  +368.921, Z    +0.000, E1    +9.337, E3 +337029.413}
SPL {X  -162.817, Y  +379.558, Z    +0.000, E1    +2.744, E3 +337029.803}
SPL {X  -162.820, Y  +384.383, Z    +0.000, E1    -0.869, E3 +337029.773}
SPL {X  -162.820, Y  +388.871, Z    +0.000, E1    -5.151, E3 +337029.479}
SPL {X  -162.820, Y  +395.861, Z    +0.000, E1   -13.028, E3 +337029.590}
SPL {X  -162.820, Y  +409.049, Z    +0.000, E1   -29.128, E3 +337028.433}
SPL {X  -162.820, Y  +444.592, Z    +0.000, E1   -49.032, E3 +337047.442}
SPL {X  -162.820, Y  +458.217, Z    +0.000, E1   -51.268, E3 +337059.388}
SPL {X  -162.820, Y  +501.848, Z    +0.000, E1   -54.235, E3 +337105.756}
ENDSPLINE

SPLINE
SPL {X  -162.820, Y  +498.156, Z    +0.000, E1   -50.986, E3 +337119.305}
ENDSPLINE

SPLINE
SPL {X  -162.820, Y  +499.429, Z    +0.000, E1   -49.453, E3 +337130.663}
SPL {X  -162.820, Y  +505.173, Z    +0.000, E1   -49.386, E3 +337141.319}
SPL {X  -162.820, Y  +510.642, Z    +0.000, E1   -49.447, E3 +337150.669}
SPL {X  -162.820, Y  +516.435, Z    +0.000, E1   -49.526, E3 +337160.547}
SPL {X  -162.820, Y  +523.383, Z    +0.000, E1   -49.407, E3 +337173.734}
SPL {X  -162.820, Y  +532.283, Z    +0.000, E1   -49.462, E3 +337189.336}
SPL {X  -162.820, Y  +541.471, Z    +0.000, E1   -49.456, E3 +337205.714}
SPL {X  -162.820, Y  +548.933, Z    +0.000, E1   -49.456, E3 +337218.903}
SPL {X  -162.820, Y  +553.997, Z    +0.000, E1   -49.325, E3 +337228.707}
SPL {X  -162.820, Y  +562.346, Z    +0.000, E1   -49.498, E3 +337242.769}
SPL {X  -162.820, Y  +570.444, Z    +0.000, E1   -49.421, E3 +337257.516}
SPL {X  -162.820, Y  +577.429, Z    +0.000, E1   -49.474, E3 +337269.630}
SPL {X  -162.820, Y  +585.965, Z    +0.000, E1   -49.447, E3 +337285.204}
SPL {X  -162.820, Y  +594.192, Z    +0.000, E1   -49.325, E3 +337300.447}
SPL {X  -162.820, Y  +600.267, Z    +0.000, E1   -49.443, E3 +337310.535}
SPL {X  -162.820, Y  +606.218, Z    +0.000, E1   -49.464, E3 +337321.082}
SPL {X  -162.820, Y  +612.538, Z    +0.000, E1   -49.488, E3 +337332.133}
SPL {X  -162.820, Y  +617.738, Z    +0.000, E1   -49.301, E3 +337342.570}
SPL {X  -162.820, Y  +624.265, Z    +0.000, E1   -49.443, E3 +337353.365}
SPL {X  -162.820, Y  +632.551, Z    +0.000, E1   -49.478, E3 +337368.134}
SPL {X  -162.820, Y  +641.207, Z    +0.000, E1   -49.420, E3 +337383.777}
SPL {X  -162.820, Y  +648.011, Z    +0.000, E1   -49.484, E3 +337395.454}
SPL {X  -162.820, Y  +655.976, Z    +0.000, E1   -49.445, E3 +337410.083}
SPL {X  -162.820, Y  +663.916, Z    +0.000, E1   -49.371, E3 +337424.512}
SPL {X  -162.820, Y  +669.755, Z    +0.000, E1   -49.387, E3 +337434.837}
SPL {X  -162.807, Y  +675.597, Z    +0.000, E1   -49.472, E3 +337444.739}
SPL {X  -162.632, Y  +681.322, Z    +0.000, E1   -49.345, E3 +337455.750}
SPL {X  -162.228, Y  +687.372, Z    +0.000, E1   -49.294, E3 +337466.837}
SPL {X  -161.723, Y  +692.372, Z    +0.000, E1   -49.172, E3 +337476.467}
SPL {X  -161.009, Y  +697.714, Z    +0.000, E1   -49.214, E3 +337485.752}
SPL {X  -160.313, Y  +701.965, Z    +0.000, E1   -48.932, E3 +337494.964}
SPL {X  -159.435, Y  +706.528, Z    +0.000, E1   -48.764, E3 +337504.091}
SPL {X  -157.894, Y  +713.249, Z    +0.000, E1   -48.586, E3 +337517.284}
SPL {X  -156.071, Y  +719.891, Z    +0.000, E1   -48.264, E3 +337530.755}
SPL {X  -154.661, Y  +724.395, Z    +0.000, E1   -47.951, E3 +337540.436}
SPL {X  -153.094, Y  +728.931, Z    +0.000, E1   -47.705, E3 +337549.873}
SPL {X  -151.300, Y  +733.655, Z    +0.000, E1   -47.339, E3 +337560.182}
SPL {X  -145.669, Y  +746.239, Z    +0.000, E1   -50.198, E3 +337566.958}
SPL {X  -135.084, Y  +764.399, Z    +0.000, E1   -44.787, E3 +337649.862}
ENDSPLINE

SPLINE
SPL {X  -153.038, Y  +729.086, Z    +0.000, E1   -30.522, E3 +337720.569}
SPL {X  -160.383, Y  +701.564, Z    +0.000, E1   -18.145, E3 +337730.605}
SPL {X  -162.078, Y  +689.023, Z    +0.000, E1   -11.510, E3 +337730.143}
SPL {X  -162.685, Y  +680.136, Z    +0.000, E1    -6.379, E3 +337730.432}
SPL {X  -162.820, Y  +672.919, Z    +0.000, E1    -1.752, E3 +337730.471}
SPL {X  -162.820, Y  +667.861, Z    +0.000, E1    +2.254, E3 +337730.272}
SPL {X  -162.820, Y  +662.755, Z    +0.000, E1    +7.521, E3 +337730.312}
SPL {X  -162.820, Y  +657.537, Z    +0.000, E1   +13.540, E3 +337729.982}
SPL {X  -162.820, Y  +650.460, Z    +0.000, E1   +22.200, E3 +337729.413}
SPL {X  -162.820, Y  +641.200, Z    +0.000, E1   +31.596, E3 +337732.037}
SPL {X  -162.820, Y  +634.978, Z    +0.000, E1   +38.045, E3 +337731.022}
SPL {X  -162.820, Y  +595.072, Z    +0.000, E1   +53.652, E3 +337752.210}
SPL {X  -162.820, Y  +560.706, Z    +0.000, E1   +50.482, E3 +337813.119}
ENDSPLINE

SPLINE
SPL {X  -162.820, Y  +562.394, Z    +0.000, E1   +48.510, E3 +337822.054}
ENDSPLINE

SPLINE
SPL {X  -162.820, Y  +555.289, Z    +0.000, E1   +48.406, E3 +337835.893}
SPL {X  -162.820, Y  +547.003, Z    +0.000, E1   +48.390, E3 +337851.306}
SPL {X  -162.820, Y  +538.900, Z    +0.000, E1   +48.334, E3 +337866.666}
SPL {X  -162.820, Y  +530.572, Z    +0.000, E1   +48.392, E3 +337881.716}
SPL {X  -162.820, Y  +522.157, Z    +0.000, E1   +48.326, E3 +337897.805}
SPL {X  -162.820, Y  +512.600, Z    +0.000, E1   +48.469, E3 +337914.581}
SPL {X  -162.820, Y  +504.728, Z    +0.000, E1   +48.342, E3 +337929.910}
ENDSPLINE

SPLINE
SPL {X  -162.820, Y  +517.326, Z    +0.000, E1   +41.232, E3 +337945.630}
ENDSPLINE

SPLINE
SPL {X  -162.820, Y  +507.007, Z    +0.000, E1   +42.470, E3 +337962.308}
SPL {X  -162.820, Y  +496.780, Z    +0.000, E1   +43.573, E3 +337978.563}
SPL {X  -162.820, Y  +487.058, Z    +0.000, E1   +44.544, E3 +337993.763}
SPL {X  -162.820, Y  +476.193, Z    +0.000, E1   +45.591, E3 +338010.202}
SPL {X  -162.820, Y  +463.464, Z    +0.000, E1   +47.025, E3 +338027.044}
SPL {X  -162.820, Y  +451.336, Z    +0.000, E1   +48.248, E3 +338042.815}
SPL {X  -162.820, Y  +440.303, Z    +0.000, E1   +49.204, E3 +338057.262}
ENDSPLINE

SPLINE
SPL {X  -162.820, Y  +446.403, Z    +0.000, E1   +44.873, E3 +338071.290}
ENDSPLINE

SPLINE
SPL {X  -162.820, Y  +437.902, Z    +0.000, E1   +44.900, E3 +338089.003}
SPL {X  -162.820, Y  +430.894, Z    +0.000, E1   +44.976, E3 +338102.989}
SPL {X  -162.820, Y  +425.053, Z    +0.000, E1   +44.824, E3 +338116.250}
SPL {X  -162.820, Y  +416.810, Z    +0.000, E1   +44.932, E3 +338132.917}
SPL {X  -162.820, Y  +408.782, Z    +0.000, E1   +44.820, E3 +338150.348}
SPL {X  -162.820, Y  +400.166, Z    +0.000, E1   +44.948, E3 +338167.651}
SPL {X  -162.820, Y  +393.279, Z    +0.000, E1   +44.825, E3 +338182.654}
SPL {X  -162.820, Y  +387.883, Z    +0.000, E1   +44.837, E3 +338193.862}
SPL {X  -162.820, Y  +382.755, Z    +0.000, E1   +44.828, E3 +338204.655}
SPL {X  -162.796, Y  +377.700, Z    +0.000, E1   +44.829, E3 +338215.235}
SPL {X  -162.619, Y  +372.412, Z    +0.000, E1   +44.928, E3 +338225.695}
SPL {X  -162.170, Y  +365.961, Z    +0.000, E1   +44.802, E3 +338240.124}
SPL {X  -161.259, Y  +358.011, Z    +0.000, E1   +44.581, E3 +338258.051}
SPL {X  -160.417, Y  +352.631, Z    +0.000, E1   +44.411, E3 +338270.066}
SPL {X  -159.536, Y  +347.962, Z    +0.000, E1   +44.302, E3 +338280.593}
SPL {X  -158.195, Y  +341.969, Z    +0.000, E1   +44.082, E3 +338294.375}
SPL {X  -156.950, Y  +337.174, Z    +0.000, E1   +43.768, E3 +338306.066}
SPL {X  -155.654, Y  +332.729, Z    +0.000, E1   +43.534, E3 +338316.708}
SPL {X  -153.067, Y  +324.996, Z    +0.000, E1   +44.257, E3 +338328.762}
SPL {X  -147.786, Y  +312.164, Z    +0.000, E1   +47.292, E3 +338337.492}
SPL {X  -142.680, Y  +302.060, Z    +0.000, E1   +42.084, E3 +338400.864}
ENDSPLINE

SPLINE
SPL {X  -151.184, Y  +320.053, Z    +0.000, E1   +32.435, E3 +338468.107}
SPL {X  -158.917, Y  +345.064, Z    +0.000, E1   +21.858, E3 +338469.456}
SPL {X  -161.350, Y  +358.672, Z    +0.000, E1   +15.089, E3 +338472.158}
SPL {X  -162.491, Y  +370.147, Z    +0.000, E1    +8.815, E3 +338475.093}
SPL {X  -162.816, Y  +379.394, Z    +0.000, E1    +3.267, E3 +338474.921}
SPL {X  -162.820, Y  +384.427, Z    +0.000, E1    -0.390, E3 +338475.441}
SPL {X  -162.820, Y  +387.736, Z    +0.000, E1    -3.142, E3 +338474.721}
SPL {X  -162.820, Y  +392.770, Z    +0.000, E1    -7.830, E3 +338475.373}
SPL {X  -162.820, Y  +398.469, Z    +0.000, E1   -14.078, E3 +338474.826}
SPL {X  -162.820, Y  +406.111, Z    +0.000, E1   -22.010, E3 +338476.006}
SPL {X  -162.820, Y  +418.653, Z    +0.000, E1   -36.657, E3 +338470.359}
SPL {X  -162.820, Y  +440.590, Z    +0.000, E1   -50.152, E3 +338475.604}
SPL {X  -162.820, Y  +447.889, Z    +0.000, E1   -43.424, E3 +338506.750}
SPL {X  -162.820, Y  +478.087, Z    +0.000, E1   -45.903, E3 +338551.969}
ENDSPLINE

SPLINE
SPL {X  -162.820, Y  +472.818, Z    +0.000, E1   -42.437, E3 +338560.910}
ENDSPLINE

SPLINE
SPL {X  -162.820, Y  +476.137, Z    +0.000, E1   -42.304, E3 +338569.324}
SPL {X  -162.820, Y  +480.895, Z    +0.000, E1   -42.223, E3 +338580.783}
SPL {X  -162.820, Y  +488.112, Z    +0.000, E1   -42.323, E3 +338596.864}
SPL {X  -162.820, Y  +496.300, Z    +0.000, E1   -42.332, E3 +338615.577}
SPL {X  -162.820, Y  +503.162, Z    +0.000, E1   -42.272, E3 +338631.494}
SPL {X  -162.820, Y  +508.157, Z    +0.000, E1   -42.280, E3 +338642.820}
SPL {X  -162.820, Y  +513.215, Z    +0.000, E1   -42.304, E3 +338654.351}
SPL {X  -162.820, Y  +518.708, Z    +0.000, E1   -42.272, E3 +338667.072}
SPL {X  -162.820, Y  +525.147, Z    +0.000, E1   -42.298, E3 +338681.815}
SPL {X  -162.820, Y  +532.723, Z    +0.000, E1   -42.344, E3 +338698.860}
SPL {X  -162.820, Y  +538.500, Z    +0.000, E1   -42.256, E3 +338712.481}
SPL {X  -162.820, Y  +542.643, Z    +0.000, E1   -42.173, E3 +338722.492}
SPL {X  -162.820, Y  +549.160, Z    +0.000, E1   -42.387, E3 +338736.250}
SPL {X  -162.820, Y  +554.884, Z    +0.000, E1   -42.207, E3 +338750.336}
SPL {X  -162.820, Y  +559.897, Z    +0.000, E1   -42.319, E3 +338761.121}
SPL {X  -162.820, Y  +565.154, Z    +0.000, E1   -42.205, E3 +338773.967}
SPL {X  -162.820, Y  +571.654, Z    +0.000, E1   -42.313, E3 +338788.179}
SPL {X  -162.820, Y  +577.246, Z    +0.000, E1   -42.284, E3 +338801.145}
SPL {X  -162.820, Y  +583.926, Z    +0.000, E1   -42.266, E3 +338816.705}
SPL {X  -162.820, Y  +589.581, Z    +0.000, E1   -42.277, E3 +338829.382}
SPL {X  -162.820, Y  +593.999, Z    +0.000, E1   -42.301, E3 +338839.433}
SPL {X  -162.820, Y  +599.194, Z    +0.000, E1   -42.235, E3 +338851.737}
SPL {X  -162.820, Y  +604.595, Z    +0.000, E1   -42.290, E3 +338863.769}
SPL {X  -162.820, Y  +609.630, Z    +0.000, E1   -42.276, E3 +338875.395}
SPL {X  -162.820, Y  +614.392, Z    +0.000, E1   -42.242, E3 +338886.495}
SPL {X  -162.820, Y  +618.928, Z    +0.000, E1   -42.220, E3 +338897.020}
SPL {X  -162.820, Y  +625.176, Z    +0.000, E1   -42.323, E3 +338910.872}
SPL {X  -162.820, Y  +630.164, Z    +0.000, E1   -42.259, E3 +338922.482}
SPL {X  -162.820, Y  +635.892, Z    +0.000, E1   -42.319, E3 +338935.474}
SPL {X  -162.820, Y  +642.066, Z    +0.000, E1   -42.247, E3 +338949.882}
SPL {X  -162.820, Y  +646.907, Z    +0.000, E1   -42.249, E3 +338961.001}
SPL {X  -162.820, Y  +652.374, Z    +0.000, E1   -42.262, E3 +338973.439}
SPL {X  -162.820, Y  +657.439, Z    +0.000, E1   -42.251, E3 +338985.112}
SPL {X  -162.820, Y  +663.328, Z    +0.000, E1   -42.283, E3 +338998.514}
SPL {X  -162.820, Y  +669.078, Z    +0.000, E1   -42.263, E3 +339011.711}
SPL {X  -162.819, Y  +673.910, Z    +0.000, E1   -42.244, E3 +339022.905}
SPL {X  -162.670, Y  +680.491, Z    +0.000, E1   -42.282, E3 +339037.947}
SPL {X  -162.151, Y  +688.243, Z    +0.000, E1   -42.207, E3 +339056.148}
SPL {X  -161.446, Y  +694.609, Z    +0.000, E1   -42.094, E3 +339071.230}
SPL {X  -160.889, Y  +698.503, Z    +0.000, E1   -41.849, E3 +339081.504}
SPL {X  -159.869, Y  +704.360, Z    +0.000, E1   -41.806, E3 +339095.446}
SPL {X  -158.502, Y  +710.748, Z    +0.000, E1   -41.532, E3 +339111.491}
SPL {X  -156.963, Y  +716.777, Z    +0.000, E1   -41.265, E3 +339126.913}
SPL {X  -155.547, Y  +721.618, Z    +0.000, E1   -40.968, E3 +339139.433}
SPL {X  -151.388, Y  +733.433, Z    +0.000, E1   -44.269, E3 +339147.136}
SPL {X  -144.352, Y  +748.818, Z    +0.000, E1   -40.701, E3 +339216.171}
SPL {X  -143.859, Y  +749.757, Z    +0.000, E1   -39.148, E3 +339244.119}
ENDSPLINE

SPLINE
SPL {X  -159.245, Y  +707.432, Z    +0.000, E1   -21.244, E3 +339276.152}
SPL {X  -162.277, Y  +686.791, Z    +0.000, E1   -10.607, E3 +339277.562}
SPL {X  -162.766, Y  +677.687, Z    +0.000, E1    -5.239, E3 +339279.752}
SPL {X  -162.820, Y  +672.396, Z    +0.000, E1    -1.801, E3 +339280.541}
SPL {X  -162.820, Y  +667.851, Z    +0.000, E1    +1.551, E3 +339280.037}
SPL {X  -162.820, Y  +664.036, Z    +0.000, E1    +4.934, E3 +339280.757}
SPL {X  -162.820, Y  +661.024, Z    +0.000, E1    +7.880, E3 +339280.026}
SPL {X  -162.820, Y  +656.051, Z    +0.000, E1   +12.848, E3 +339280.894}
SPL {X  -162.820, Y  +650.794, Z    +0.000, E1   +18.580, E3 +339280.450}
SPL {X  -162.820, Y  +638.947, Z    +0.000, E1   +31.033, E3 +339278.797}
SPL {X  -162.820, Y  +608.150, Z    +0.000, E1   +43.921, E3 +339305.030}
SPL {X  -162.820, Y  +574.255, Z    +0.000, E1   +46.562, E3 +339354.824}
ENDSPLINE

SPLINE
SPL {X  -162.820, Y  +579.440, Z    +0.000, E1   +42.450, E3 +339368.012}
ENDSPLINE

SPLINE
SPL {X  -162.820, Y  +573.350, Z    +0.000, E1   +42.340, E3 +339382.689}
SPL {X  -162.820, Y  +565.899, Z    +0.000, E1   +42.413, E3 +339399.273}
SPL {X  -162.820, Y  +560.278, Z    +0.000, E1   +42.308, E3 +339412.610}
SPL {X  -162.820, Y  +554.421, Z    +0.000, E1   +42.414, E3 +339425.478}
SPL {X  -162.820, Y  +547.774, Z    +0.000, E1   +42.344, E3 +339441.051}
SPL {X  -162.820, Y  +541.056, Z    +0.000, E1   +42.452, E3 +339455.713}
SPL {X  -162.820, Y  +535.223, Z    +0.000, E1   +42.386, E3 +339469.407}
SPL {X  -162.820, Y  +529.084, Z    +0.000, E1   +42.400, E3 +339483.330}
SPL {X  -162.820, Y  +524.911, Z    +0.000, E1   +42.325, E3 +339493.176}
SPL {X  -162.820, Y  +519.984, Z    +0.000, E1   +42.385, E3 +339504.246}
SPL {X  -162.820, Y  +512.536, Z    +0.000, E1   +42.385, E3 +339521.357}
SPL {X  -162.820, Y  +505.746, Z    +0.000, E1   +42.400, E3 +339536.601}
SPL {X  -162.820, Y  +500.461, Z    +0.000, E1   +42.387, E3 +339548.728}
SPL {X  -162.820, Y  +494.841, Z    +0.000, E1   +42.316, E3 +339562.055}
SPL {X  -162.820, Y  +486.958, Z    +0.000, E1   +42.460, E3 +339579.347}
SPL {X  -162.820, Y  +464.528, Z    +0.000, E1   +47.611, E3 +339595.561}
SPL {X  -162.820, Y  +458.830, Z    +0.000, E1   +46.994, E3 +339610.239}
SPL {X  -162.820, Y  +455.537, Z    +0.000, E1   +45.900, E3 +339623.058}
SPL {X  -162.820, Y  +452.032, Z    +0.000, E1   +45.224, E3 +339634.263}
SPL {X  -162.820, Y  +446.617, Z    +0.000, E1   +44.768, E3 +339648.349}
SPL {X  -162.820, Y  +440.464, Z    +0.000, E1   +44.845, E3 +339660.651}
SPL {X  -162.820, Y  +435.902, Z    +0.000, E1   +44.853, E3 +339670.174}
SPL {X  -162.820, Y  +429.336, Z    +0.000, E1   +44.917, E3 +339683.693}
SPL {X  -162.820, Y  +423.193, Z    +0.000, E1   +44.819, E3 +339696.952}
SPL {X  -162.820, Y  +418.403, Z    +0.000, E1   +44.941, E3 +339706.287}
SPL {X  -162.820, Y  +412.479, Z    +0.000, E1   +44.780, E3 +339719.717}
SPL {X  -162.820, Y  +406.707, Z    +0.000, E1   +44.849, E3 +339731.290}
SPL {X  -162.820, Y  +400.166, Z    +0.000, E1   +44.948, E3 +339744.574}
SPL {X  -162.820, Y  +393.279, Z    +0.000, E1   +44.825, E3 +339759.577}
SPL {X  -162.820, Y  +387.883, Z    +0.000, E1   +44.837, E3 +339770.785}
SPL {X  -162.820, Y  +382.755, Z    +0.000, E1   +44.828, E3 +339781.578}
SPL {X  -162.796, Y  +377.700, Z    +0.000, E1   +44.829, E3 +339792.158}
SPL {X  -162.619, Y  +372.412, Z    +0.000, E1   +44.928, E3 +339802.618}
SPL {X  -162.311, Y  +367.633, Z    +0.000, E1   +44.798, E3 +339813.385}
SPL {X  -161.766, Y  +362.002, Z    +0.000, E1   +44.644, E3 +339826.144}
SPL {X  -161.043, Y  +356.508, Z    +0.000, E1   +44.528, E3 +339838.258}
SPL {X  -160.417, Y  +352.631, Z    +0.000, E1   +44.411, E3 +339846.989}
SPL {X  -159.536, Y  +347.962, Z    +0.000, E1   +44.302, E3 +339857.516}
SPL {X  -158.195, Y  +341.969, Z    +0.000, E1   +44.082, E3 +339871.298}
SPL {X  -156.950, Y  +337.174, Z    +0.000, E1   +43.768, E3 +339882.989}
SPL {X  -155.654, Y  +332.729, Z    +0.000, E1   +43.534, E3 +339893.631}
SPL {X  -154.189, Y  +328.191, Z    +0.000, E1   +43.338, E3 +339904.127}
SPL {X  -149.333, Y  +315.614, Z    +0.000, E1   +46.650, E3 +339911.443}
SPL {X  -142.680, Y  +302.060, Z    +0.000, E1   +42.084, E3 +339977.787}
ENDSPLINE

SPLINE
SPL {X  -151.184, Y  +320.053, Z    +0.000, E1   +32.435, E3 +340045.030}
SPL {X  -158.917, Y  +345.064, Z    +0.000, E1   +21.858, E3 +340046.379}
SPL {X  -161.350, Y  +358.672, Z    +0.000, E1   +15.089, E3 +340049.082}
SPL {X  -162.491, Y  +370.147, Z    +0.000, E1    +8.815, E3 +340052.016}
SPL {X  -162.771, Y  +376.522, Z    +0.000, E1    +5.005, E3 +340051.625}
SPL {X  -162.820, Y  +383.029, Z    +0.000, E1    +0.769, E3 +340052.193}
SPL {X  -162.820, Y  +387.736, Z    +0.000, E1    -3.142, E3 +340051.644}
SPL {X  -162.820, Y  +391.456, Z    +0.000, E1    -6.603, E3 +340052.431}
SPL {X  -162.820, Y  +397.032, Z    +0.000, E1   -12.435, E3 +340051.878}
SPL {X  -162.820, Y  +406.111, Z    +0.000, E1   -22.010, E3 +340052.929}
SPL {X  -162.820, Y  +418.653, Z    +0.000, E1   -36.657, E3 +340047.282}
SPL {X  -162.820, Y  +440.590, Z    +0.000, E1   -50.152, E3 +340052.528}
SPL {X  -162.820, Y  +447.889, Z    +0.000, E1   -43.424, E3 +340083.673}
SPL {X  -162.820, Y  +478.087, Z    +0.000, E1   -45.903, E3 +340128.892}
ENDSPLINE

SPLINE
SPL {X  -162.820, Y  +474.900, Z    +0.000, E1   -42.394, E3 +340143.045}
ENDSPLINE

SPLINE
SPL {X  -162.820, Y  +480.895, Z    +0.000, E1   -42.223, E3 +340157.707}
SPL {X  -162.820, Y  +485.782, Z    +0.000, E1   -42.348, E3 +340168.052}
SPL {X  -162.820, Y  +489.480, Z    +0.000, E1   -42.230, E3 +340177.279}
SPL {X  -162.820, Y  +496.300, Z    +0.000, E1   -42.332, E3 +340192.500}
SPL {X  -162.820, Y  +503.162, Z    +0.000, E1   -42.272, E3 +340208.417}
SPL {X  -162.820, Y  +509.376, Z    +0.000, E1   -42.304, E3 +340222.508}
SPL {X  -162.820, Y  +514.403, Z    +0.000, E1   -42.285, E3 +340234.003}
SPL {X  -162.820, Y  +520.311, Z    +0.000, E1   -42.317, E3 +340247.572}
SPL {X  -162.820, Y  +526.529, Z    +0.000, E1   -42.247, E3 +340262.042}
SPL {X  -162.820, Y  +531.715, Z    +0.000, E1   -42.312, E3 +340273.564}
SPL {X  -162.820, Y  +537.459, Z    +0.000, E1   -42.308, E3 +340286.823}
SPL {X  -162.820, Y  +542.643, Z    +0.000, E1   -42.173, E3 +340299.415}
SPL {X  -162.820, Y  +549.160, Z    +0.000, E1   -42.387, E3 +340313.173}
SPL {X  -162.820, Y  +554.884, Z    +0.000, E1   -42.207, E3 +340327.259}
SPL {X  -162.820, Y  +561.114, Z    +0.000, E1   -42.336, E3 +340340.839}
SPL {X  -162.820, Y  +566.097, Z    +0.000, E1   -42.118, E3 +340353.449}
SPL {X  -162.820, Y  +571.654, Z    +0.000, E1   -42.313, E3 +340365.103}
SPL {X  -162.820, Y  +577.246, Z    +0.000, E1   -42.284, E3 +340378.068}
SPL {X  -162.820, Y  +583.926, Z    +0.000, E1   -42.266, E3 +340393.628}
SPL {X  -162.820, Y  +589.581, Z    +0.000, E1   -42.277, E3 +340406.305}
SPL {X  -162.820, Y  +593.999, Z    +0.000, E1   -42.301, E3 +340416.356}
SPL {X  -162.820, Y  +599.194, Z    +0.000, E1   -42.235, E3 +340428.660}
SPL {X  -162.820, Y  +604.595, Z    +0.000, E1   -42.290, E3 +340440.692}
SPL {X  -162.820, Y  +609.630, Z    +0.000, E1   -42.276, E3 +340452.318}
SPL {X  -162.820, Y  +614.392, Z    +0.000, E1   -42.242, E3 +340463.418}
SPL {X  -162.820, Y  +620.424, Z    +0.000, E1   -42.277, E3 +340477.166}
SPL {X  -162.820, Y  +626.430, Z    +0.000, E1   -42.291, E3 +340490.715}
SPL {X  -162.820, Y  +631.865, Z    +0.000, E1   -42.327, E3 +340503.009}
SPL {X  -162.820, Y  +637.189, Z    +0.000, E1   -42.236, E3 +340515.683}
SPL {X  -162.820, Y  +642.066, Z    +0.000, E1   -42.247, E3 +340526.805}
SPL {X  -162.820, Y  +646.907, Z    +0.000, E1   -42.249, E3 +340537.924}
SPL {X  -162.820, Y  +652.374, Z    +0.000, E1   -42.262, E3 +340550.362}
SPL {X  -162.820, Y  +657.439, Z    +0.000, E1   -42.251, E3 +340562.035}
SPL {X  -162.820, Y  +663.328, Z    +0.000, E1   -42.283, E3 +340575.437}
SPL {X  -162.820, Y  +669.078, Z    +0.000, E1   -42.263, E3 +340588.634}
SPL {X  -162.819, Y  +673.910, Z    +0.000, E1   -42.244, E3 +340599.828}
SPL {X  -162.729, Y  +678.944, Z    +0.000, E1   -42.273, E3 +340611.195}
SPL {X  -162.479, Y  +684.035, Z    +0.000, E1   -42.168, E3 +340623.533}
SPL {X  -162.026, Y  +689.560, Z    +0.000, E1   -42.192, E3 +340636.021}
SPL {X  -161.446, Y  +694.609, Z    +0.000, E1   -42.094, E3 +340648.153}
SPL {X  -160.681, Y  +699.806, Z    +0.000, E1   -41.866, E3 +340661.436}
SPL {X  -159.658, Y  +705.434, Z    +0.000, E1   -41.735, E3 +340675.066}
SPL {X  -158.727, Y  +709.780, Z    +0.000, E1   -41.560, E3 +340685.934}
SPL {X  -157.709, Y  +713.973, Z    +0.000, E1   -41.360, E3 +340696.788}
SPL {X  -156.530, Y  +718.319, Z    +0.000, E1   -41.164, E3 +340707.732}
SPL {X  -155.547, Y  +721.618, Z    +0.000, E1   -40.968, E3 +340716.356}
SPL {X  -151.388, Y  +733.433, Z    +0.000, E1   -44.269, E3 +340724.059}
SPL {X  -144.352, Y  +748.818, Z    +0.000, E1   -40.701, E3 +340793.094}
SPL {X  -143.859, Y  +749.757, Z    +0.000, E1   -39.148, E3 +340821.042}
ENDSPLINE

SPLINE
SPL {X  -159.245, Y  +707.432, Z    +0.000, E1   -21.244, E3 +340853.075}
SPL {X  -162.277, Y  +686.791, Z    +0.000, E1   -10.607, E3 +340854.485}
SPL {X  -162.766, Y  +677.687, Z    +0.000, E1    -5.239, E3 +340856.675}
SPL {X  -162.820, Y  +672.396, Z    +0.000, E1    -1.801, E3 +340857.464}
SPL {X  -162.820, Y  +667.851, Z    +0.000, E1    +1.551, E3 +340856.960}
SPL {X  -162.820, Y  +664.036, Z    +0.000, E1    +4.934, E3 +340857.680}
SPL {X  -162.820, Y  +661.024, Z    +0.000, E1    +7.880, E3 +340856.949}
SPL {X  -162.820, Y  +656.051, Z    +0.000, E1   +12.848, E3 +340857.817}
SPL {X  -162.820, Y  +650.794, Z    +0.000, E1   +18.580, E3 +340857.373}
SPL {X  -162.820, Y  +638.947, Z    +0.000, E1   +31.033, E3 +340855.720}
SPL {X  -162.820, Y  +608.150, Z    +0.000, E1   +43.921, E3 +340881.953}
SPL {X  -162.820, Y  +574.255, Z    +0.000, E1   +46.562, E3 +340931.747}
ENDSPLINE

SPLINE
SPL {X  -162.820, Y  +579.440, Z    +0.000, E1   +42.450, E3 +340944.935}
ENDSPLINE

SPLINE
SPL {X  -162.820, Y  +573.350, Z    +0.000, E1   +42.340, E3 +340959.612}
SPL {X  -162.820, Y  +565.899, Z    +0.000, E1   +42.413, E3 +340976.196}
SPL {X  -162.820, Y  +560.278, Z    +0.000, E1   +42.308, E3 +340989.533}
SPL {X  -162.820, Y  +554.421, Z    +0.000, E1   +42.414, E3 +341002.401}
SPL {X  -162.820, Y  +547.774, Z    +0.000, E1   +42.344, E3 +341017.974}
SPL {X  -162.820, Y  +541.056, Z    +0.000, E1   +42.452, E3 +341032.636}
SPL {X  -162.820, Y  +535.223, Z    +0.000, E1   +42.386, E3 +341046.330}
SPL {X  -162.820, Y  +529.084, Z    +0.000, E1   +42.400, E3 +341060.253}
SPL {X  -162.820, Y  +524.911, Z    +0.000, E1   +42.325, E3 +341070.099}
SPL {X  -162.820, Y  +519.984, Z    +0.000, E1   +42.385, E3 +341081.169}
SPL {X  -162.820, Y  +514.684, Z    +0.000, E1   +42.289, E3 +341093.741}
SPL {X  -162.820, Y  +508.859, Z    +0.000, E1   +42.416, E3 +341106.392}
SPL {X  -162.820, Y  +501.651, Z    +0.000, E1   +42.423, E3 +341122.868}
SPL {X  -162.820, Y  +496.578, Z    +0.000, E1   +42.329, E3 +341134.776}
SPL {X  -162.820, Y  +491.918, Z    +0.000, E1   +42.382, E3 +341145.269}
SPL {X  -162.820, Y  +485.695, Z    +0.000, E1   +42.386, E3 +341159.407}
SPL {X  -162.820, Y  +464.528, Z    +0.000, E1   +47.611, E3 +341172.484}
SPL {X  -162.820, Y  +459.899, Z    +0.000, E1   +47.097, E3 +341184.327}
SPL {X  -162.820, Y  +455.990, Z    +0.000, E1   +46.212, E3 +341197.400}
SPL {X  -162.820, Y  +452.032, Z    +0.000, E1   +45.224, E3 +341211.186}
SPL {X  -162.820, Y  +446.617, Z    +0.000, E1   +44.768, E3 +341225.272}
SPL {X  -162.820, Y  +437.902, Z    +0.000, E1   +44.900, E3 +341242.849}
SPL {X  -162.820, Y  +430.894, Z    +0.000, E1   +44.976, E3 +341256.835}
SPL {X  -162.820, Y  +425.053, Z    +0.000, E1   +44.824, E3 +341270.097}
SPL {X  -162.820, Y  +418.403, Z    +0.000, E1   +44.941, E3 +341283.210}
SPL {X  -162.820, Y  +412.479, Z    +0.000, E1   +44.780, E3 +341296.640}
SPL {X  -162.820, Y  +406.707, Z    +0.000, E1   +44.849, E3 +341308.213}
SPL {X  -162.820, Y  +401.619, Z    +0.000, E1   +44.978, E3 +341318.115}
SPL {X  -162.820, Y  +394.771, Z    +0.000, E1   +44.856, E3 +341333.354}
SPL {X  -162.820, Y  +387.883, Z    +0.000, E1   +44.837, E3 +341347.708}
SPL {X  -162.820, Y  +382.755, Z    +0.000, E1   +44.828, E3 +341358.501}
SPL {X  -162.796, Y  +377.700, Z    +0.000, E1   +44.829, E3 +341369.081}
SPL {X  -162.619, Y  +372.412, Z    +0.000, E1   +44.928, E3 +341379.541}
SPL {X  -162.311, Y  +367.633, Z    +0.000, E1   +44.798, E3 +341390.308}
SPL {X  -161.766, Y  +362.002, Z    +0.000, E1   +44.644, E3 +341403.067}
SPL {X  -161.043, Y  +356.508, Z    +0.000, E1   +44.528, E3 +341415.181}
SPL {X  -160.417, Y  +352.631, Z    +0.000, E1   +44.411, E3 +341423.912}
SPL {X  -159.536, Y  +347.962, Z    +0.000, E1   +44.302, E3 +341434.439}
SPL {X  -158.195, Y  +341.969, Z    +0.000, E1   +44.082, E3 +341448.221}
SPL {X  -156.950, Y  +337.174, Z    +0.000, E1   +43.768, E3 +341459.912}
SPL {X  -155.654, Y  +332.729, Z    +0.000, E1   +43.534, E3 +341470.554}
SPL {X  -153.067, Y  +324.996, Z    +0.000, E1   +44.257, E3 +341482.608}
SPL {X  -147.786, Y  +312.164, Z    +0.000, E1   +47.292, E3 +341491.338}
SPL {X  -142.680, Y  +302.060, Z    +0.000, E1   +42.084, E3 +341554.710}
ENDSPLINE

SPLINE
SPL {X  -151.184, Y  +320.053, Z    +0.000, E1   +32.435, E3 +341621.954}
SPL {X  -158.917, Y  +345.064, Z    +0.000, E1   +21.858, E3 +341623.302}
SPL {X  -161.350, Y  +358.672, Z    +0.000, E1   +15.089, E3 +341626.005}
SPL {X  -162.491, Y  +370.147, Z    +0.000, E1    +8.815, E3 +341628.939}
SPL {X  -162.816, Y  +379.394, Z    +0.000, E1    +3.267, E3 +341628.767}
SPL {X  -162.820, Y  +384.427, Z    +0.000, E1    -0.390, E3 +341629.287}
SPL {X  -162.820, Y  +387.736, Z    +0.000, E1    -3.142, E3 +341628.567}
SPL {X  -162.820, Y  +392.770, Z    +0.000, E1    -7.830, E3 +341629.219}
SPL {X  -162.820, Y  +398.469, Z    +0.000, E1   -14.078, E3 +341628.672}
SPL {X  -162.820, Y  +406.111, Z    +0.000, E1   -22.010, E3 +341629.852}
SPL {X  -162.820, Y  +418.653, Z    +0.000, E1   -36.657, E3 +341624.205}
SPL {X  -162.820, Y  +440.590, Z    +0.000, E1   -50.152, E3 +341629.451}
SPL {X  -162.820, Y  +447.889, Z    +0.000, E1   -43.424, E3 +341660.596}
SPL {X  -162.820, Y  +479.020, Z    +0.000, E1   -47.189, E3 +341700.173}
ENDSPLINE

SPLINE
SPL {X  -162.820, Y  +474.886, Z    +0.000, E1   -43.721, E3 +341712.057}
ENDSPLINE

SPLINE
SPL {X  -162.820, Y  +477.319, Z    +0.000, E1   -42.306, E3 +341725.983}
SPL {X  -162.820, Y  +483.923, Z    +0.000, E1   -42.291, E3 +341741.190}
SPL {X  -162.820, Y  +489.480, Z    +0.000, E1   -42.230, E3 +341754.202}
SPL {X  -162.820, Y  +494.825, Z    +0.000, E1   -42.287, E3 +341766.150}
SPL {X  -162.820, Y  +501.023, Z    +0.000, E1   -42.347, E3 +341780.032}
SPL {X  -162.820, Y  +506.968, Z    +0.000, E1   -42.248, E3 +341794.223}
SPL {X  -162.820, Y  +513.215, Z    +0.000, E1   -42.304, E3 +341808.197}
SPL {X  -162.820, Y  +518.708, Z    +0.000, E1   -42.272, E3 +341820.919}
SPL {X  -162.820, Y  +525.147, Z    +0.000, E1   -42.298, E3 +341835.661}
SPL {X  -162.820, Y  +531.715, Z    +0.000, E1   -42.312, E3 +341850.487}
SPL {X  -162.820, Y  +537.459, Z    +0.000, E1   -42.308, E3 +341863.746}
SPL {X  -162.820, Y  +542.643, Z    +0.000, E1   -42.173, E3 +341876.338}
SPL {X  -162.820, Y  +549.160, Z    +0.000, E1   -42.387, E3 +341890.096}
SPL {X  -162.820, Y  +554.884, Z    +0.000, E1   -42.207, E3 +341904.182}
SPL {X  -162.820, Y  +561.114, Z    +0.000, E1   -42.336, E3 +341917.762}
SPL {X  -162.820, Y  +566.097, Z    +0.000, E1   -42.118, E3 +341930.372}
SPL {X  -162.820, Y  +571.654, Z    +0.000, E1   -42.313, E3 +341942.026}
SPL {X  -162.820, Y  +577.246, Z    +0.000, E1   -42.284, E3 +341954.991}
SPL {X  -162.820, Y  +582.233, Z    +0.000, E1   -42.188, E3 +341966.970}
SPL {X  -162.820, Y  +588.138, Z    +0.000, E1   -42.308, E3 +341979.869}
SPL {X  -162.820, Y  +593.999, Z    +0.000, E1   -42.301, E3 +341993.279}
SPL {X  -162.820, Y  +599.194, Z    +0.000, E1   -42.235, E3 +342005.584}
SPL {X  -162.820, Y  +604.595, Z    +0.000, E1   -42.290, E3 +342017.615}
SPL {X  -162.820, Y  +609.630, Z    +0.000, E1   -42.276, E3 +342029.241}
SPL {X  -162.820, Y  +614.392, Z    +0.000, E1   -42.242, E3 +342040.341}
SPL {X  -162.820, Y  +620.424, Z    +0.000, E1   -42.277, E3 +342054.089}
SPL {X  -162.820, Y  +626.430, Z    +0.000, E1   -42.291, E3 +342067.638}
SPL {X  -162.820, Y  +631.865, Z    +0.000, E1   -42.327, E3 +342079.932}
SPL {X  -162.820, Y  +637.189, Z    +0.000, E1   -42.236, E3 +342092.606}
SPL {X  -162.820, Y  +642.066, Z    +0.000, E1   -42.247, E3 +342103.728}
SPL {X  -162.820, Y  +646.907, Z    +0.000, E1   -42.249, E3 +342114.847}
SPL {X  -162.820, Y  +652.374, Z    +0.000, E1   -42.262, E3 +342127.286}
SPL {X  -162.820, Y  +658.634, Z    +0.000, E1   -42.281, E3 +342141.643}
SPL {X  -162.820, Y  +664.480, Z    +0.000, E1   -42.257, E3 +342155.037}
SPL {X  -162.820, Y  +669.078, Z    +0.000, E1   -42.263, E3 +342165.557}
SPL {X  -162.819, Y  +673.910, Z    +0.000, E1   -42.244, E3 +342176.751}
SPL {X  -162.729, Y  +678.944, Z    +0.000, E1   -42.273, E3 +342188.119}
SPL {X  -162.479, Y  +684.035, Z    +0.000, E1   -42.168, E3 +342200.456}
SPL {X  -162.026, Y  +689.560, Z    +0.000, E1   -42.192, E3 +342212.945}
SPL {X  -161.446, Y  +694.609, Z    +0.000, E1   -42.094, E3 +342225.077}
SPL {X  -160.681, Y  +699.806, Z    +0.000, E1   -41.866, E3 +342238.360}
SPL {X  -159.658, Y  +705.434, Z    +0.000, E1   -41.735, E3 +342251.990}
SPL {X  -158.502, Y  +710.748, Z    +0.000, E1   -41.532, E3 +342265.337}
SPL {X  -157.452, Y  +714.962, Z    +0.000, E1   -41.276, E3 +342276.332}
SPL {X  -156.530, Y  +718.319, Z    +0.000, E1   -41.164, E3 +342284.655}
SPL {X  -155.547, Y  +721.618, Z    +0.000, E1   -40.968, E3 +342293.279}
SPL {X  -151.388, Y  +733.433, Z    +0.000, E1   -44.269, E3 +342300.982}
SPL {X  -144.352, Y  +748.818, Z    +0.000, E1   -40.701, E3 +342370.017}
SPL {X  -143.859, Y  +749.757, Z    +0.000, E1   -39.148, E3 +342397.965}
ENDSPLINE

SPLINE
SPL {X  -159.245, Y  +707.432, Z    +0.000, E1   -21.244, E3 +342429.998}
SPL {X  -162.277, Y  +686.791, Z    +0.000, E1   -10.607, E3 +342431.408}
SPL {X  -162.766, Y  +677.687, Z    +0.000, E1    -5.239, E3 +342433.598}
SPL {X  -162.820, Y  +671.059, Z    +0.000, E1    -0.934, E3 +342433.954}
SPL {X  -162.820, Y  +666.960, Z    +0.000, E1    +2.343, E3 +342434.231}
SPL {X  -162.820, Y  +662.610, Z    +0.000, E1    +6.209, E3 +342434.257}
SPL {X  -162.820, Y  +654.280, Z    +0.000, E1   +14.617, E3 +342434.590}
SPL {X  -162.820, Y  +638.947, Z    +0.000, E1   +31.033, E3 +342432.643}
SPL {X  -162.820, Y  +608.150, Z    +0.000, E1   +43.921, E3 +342458.876}
SPL {X  -162.820, Y  +574.255, Z    +0.000, E1   +46.562, E3 +342508.670}
ENDSPLINE

SPLINE
SPL {X  -162.820, Y  +579.440, Z    +0.000, E1   +42.450, E3 +342521.858}
ENDSPLINE

SPLINE
SPL {X  -162.820, Y  +574.443, Z    +0.000, E1   +42.333, E3 +342533.952}
SPL {X  -162.820, Y  +568.554, Z    +0.000, E1   +42.362, E3 +342547.315}
SPL {X  -162.820, Y  +561.474, Z    +0.000, E1   +42.369, E3 +342563.500}
SPL {X  -162.820, Y  +554.421, Z    +0.000, E1   +42.414, E3 +342579.324}
SPL {X  -162.820, Y  +547.774, Z    +0.000, E1   +42.344, E3 +342594.898}
SPL {X  -162.820, Y  +541.056, Z    +0.000, E1   +42.452, E3 +342609.559}
SPL {X  -162.820, Y  +535.223, Z    +0.000, E1   +42.386, E3 +342623.253}
SPL {X  -162.820, Y  +529.084, Z    +0.000, E1   +42.400, E3 +342637.176}
SPL {X  -162.820, Y  +522.568, Z    +0.000, E1   +42.385, E3 +342652.205}
SPL {X  -162.820, Y  +515.708, Z    +0.000, E1   +42.333, E3 +342668.173}
SPL {X  -162.820, Y  +508.859, Z    +0.000, E1   +42.416, E3 +342683.315}
SPL {X  -162.820, Y  +501.651, Z    +0.000, E1   +42.423, E3 +342699.791}
SPL {X  -162.820, Y  +494.841, Z    +0.000, E1   +42.316, E3 +342715.901}
SPL {X  -162.820, Y  +486.958, Z    +0.000, E1   +42.460, E3 +342733.194}
SPL {X  -162.820, Y  +466.305, Z    +0.000, E1   +47.564, E3 +342746.201}
SPL {X  -162.820, Y  +460.790, Z    +0.000, E1   +47.323, E3 +342758.376}
SPL {X  -162.820, Y  +455.990, Z    +0.000, E1   +46.212, E3 +342774.324}
SPL {X  -162.820, Y  +452.032, Z    +0.000, E1   +45.224, E3 +342788.109}
SPL {X  -162.820, Y  +446.617, Z    +0.000, E1   +44.768, E3 +342802.195}
SPL {X  -162.820, Y  +437.902, Z    +0.000, E1   +44.900, E3 +342819.772}
SPL {X  -162.820, Y  +430.894, Z    +0.000, E1   +44.976, E3 +342833.758}
SPL {X  -162.820, Y  +425.053, Z    +0.000, E1   +44.824, E3 +342847.020}
SPL {X  -162.820, Y  +416.810, Z    +0.000, E1   +44.932, E3 +342863.686}
SPL {X  -162.820, Y  +408.782, Z    +0.000, E1   +44.820, E3 +342881.117}
SPL {X  -162.820, Y  +401.619, Z    +0.000, E1   +44.978, E3 +342895.038}
SPL {X  -162.820, Y  +394.771, Z    +0.000, E1   +44.856, E3 +342910.277}
SPL {X  -162.820, Y  +387.883, Z    +0.000, E1   +44.837, E3 +342924.631}
SPL {X  -162.820, Y  +382.755, Z    +0.000, E1   +44.828, E3 +342935.424}
SPL {X  -162.796, Y  +377.700, Z    +0.000, E1   +44.829, E3 +342946.004}
SPL {X  -162.619, Y  +372.412, Z    +0.000, E1   +44.928, E3 +342956.464}
SPL {X  -162.311, Y  +367.633, Z    +0.000, E1   +44.798, E3 +342967.231}
SPL {X  -161.766, Y  +362.002, Z    +0.000, E1   +44.644, E3 +342979.990}
SPL {X  -161.043, Y  +356.508, Z    +0.000, E1   +44.528, E3 +342992.104}
SPL {X  -160.070, Y  +350.699, Z    +0.000, E1   +44.409, E3 +343005.056}
SPL {X  -158.853, Y  +344.776, Z    +0.000, E1   +44.148, E3 +343018.877}
SPL {X  -157.292, Y  +338.433, Z    +0.000, E1   +43.917, E3 +343033.555}
SPL {X  -155.654, Y  +332.729, Z    +0.000, E1   +43.534, E3 +343047.477}
SPL {X  -154.189, Y  +328.191, Z    +0.000, E1   +43.338, E3 +343057.973}
SPL {X  -149.333, Y  +315.614, Z    +0.000, E1   +46.650, E3 +343065.289}
SPL {X  -142.680, Y  +302.060, Z    +0.000, E1   +42.084, E3 +343131.634}
ENDSPLINE

SPLINE
SPL {X  -151.184, Y  +320.053, Z    +0.000, E1   +32.435, E3 +343198.877}
SPL {X  -158.917, Y  +345.064, Z    +0.000, E1   +21.858, E3 +343200.225}
SPL {X  -161.350, Y  +358.672, Z    +0.000, E1   +15.089, E3 +343202.928}
SPL {X  -162.491, Y  +370.147, Z    +0.000, E1    +8.815, E3 +343205.862}
SPL {X  -162.771, Y  +376.522, Z    +0.000, E1    +5.005, E3 +343205.472}
SPL {X  -162.820, Y  +383.029, Z    +0.000, E1    +0.769, E3 +343206.039}
SPL {X  -162.820, Y  +387.736, Z    +0.000, E1    -3.142, E3 +343205.490}
SPL {X  -162.820, Y  +392.770, Z    +0.000, E1    -7.830, E3 +343206.142}
SPL {X  -162.820, Y  +398.469, Z    +0.000, E1   -14.078, E3 +343205.595}
SPL {X  -162.820, Y  +406.111, Z    +0.000, E1   -22.010, E3 +343206.775}
SPL {X  -162.820, Y  +418.653, Z    +0.000, E1   -36.657, E3 +343201.128}
SPL {X  -162.820, Y  +440.590, Z    +0.000, E1   -50.152, E3 +343206.374}
SPL {X  -162.820, Y  +447.889, Z    +0.000, E1   -43.424, E3 +343237.520}
SPL {X  -162.820, Y  +478.087, Z    +0.000, E1   -45.903, E3 +343282.739}
ENDSPLINE

SPLINE
SPL {X  -162.820, Y  +474.900, Z    +0.000, E1   -42.394, E3 +343296.891}
ENDSPLINE

SPLINE
SPL {X  -162.820, Y  +480.895, Z    +0.000, E1   -42.223, E3 +343311.553}
SPL {X  -162.820, Y  +485.782, Z    +0.000, E1   -42.348, E3 +343321.898}
SPL {X  -162.820, Y  +489.480, Z    +0.000, E1   -42.230, E3 +343331.125}
SPL {X  -162.820, Y  +494.825, Z    +0.000, E1   -42.287, E3 +343343.073}
SPL {X  -162.820, Y  +501.023, Z    +0.000, E1   -42.347, E3 +343356.955}
SPL {X  -162.820, Y  +506.968, Z    +0.000, E1   -42.248, E3 +343371.146}
SPL {X  -162.820, Y  +513.215, Z    +0.000, E1   -42.304, E3 +343385.120}
SPL {X  -162.820, Y  +518.708, Z    +0.000, E1   -42.272, E3 +343397.842}
SPL {X  -162.820, Y  +525.147, Z    +0.000, E1   -42.298, E3 +343412.584}
SPL {X  -162.820, Y  +531.715, Z    +0.000, E1   -42.312, E3 +343427.410}
SPL {X  -162.820, Y  +537.459, Z    +0.000, E1   -42.308, E3 +343440.669}
SPL {X  -162.820, Y  +542.643, Z    +0.000, E1   -42.173, E3 +343453.261}
SPL {X  -162.820, Y  +549.160, Z    +0.000, E1   -42.387, E3 +343467.019}
SPL {X  -162.820, Y  +554.884, Z    +0.000, E1   -42.207, E3 +343481.105}
SPL {X  -162.820, Y  +561.114, Z    +0.000, E1   -42.336, E3 +343494.685}
SPL {X  -162.820, Y  +566.097, Z    +0.000, E1   -42.118, E3 +343507.296}
SPL {X  -162.820, Y  +571.654, Z    +0.000, E1   -42.313, E3 +343518.949}
SPL {X  -162.820, Y  +577.246, Z    +0.000, E1   -42.284, E3 +343531.914}
SPL {X  -162.820, Y  +582.233, Z    +0.000, E1   -42.188, E3 +343543.893}
SPL {X  -162.820, Y  +588.138, Z    +0.000, E1   -42.308, E3 +343556.792}
SPL {X  -162.820, Y  +593.999, Z    +0.000, E1   -42.301, E3 +343570.202}
SPL {X  -162.820, Y  +599.194, Z    +0.000, E1   -42.235, E3 +343582.507}
SPL {X  -162.820, Y  +604.595, Z    +0.000, E1   -42.290, E3 +343594.538}
SPL {X  -162.820, Y  +609.630, Z    +0.000, E1   -42.276, E3 +343606.164}
SPL {X  -162.820, Y  +614.392, Z    +0.000, E1   -42.242, E3 +343617.264}
SPL {X  -162.820, Y  +620.424, Z    +0.000, E1   -42.277, E3 +343631.012}
SPL {X  -162.820, Y  +626.430, Z    +0.000, E1   -42.291, E3 +343644.561}
SPL {X  -162.820, Y  +631.865, Z    +0.000, E1   -42.327, E3 +343656.855}
SPL {X  -162.820, Y  +637.189, Z    +0.000, E1   -42.236, E3 +343669.529}
SPL {X  -162.820, Y  +642.066, Z    +0.000, E1   -42.247, E3 +343680.651}
SPL {X  -162.820, Y  +646.907, Z    +0.000, E1   -42.249, E3 +343691.770}
SPL {X  -162.820, Y  +652.374, Z    +0.000, E1   -42.262, E3 +343704.209}
SPL {X  -162.820, Y  +657.439, Z    +0.000, E1   -42.251, E3 +343715.882}
SPL {X  -162.820, Y  +663.328, Z    +0.000, E1   -42.283, E3 +343729.284}
SPL {X  -162.820, Y  +669.078, Z    +0.000, E1   -42.263, E3 +343742.480}
SPL {X  -162.819, Y  +673.910, Z    +0.000, E1   -42.244, E3 +343753.674}
SPL {X  -162.729, Y  +678.944, Z    +0.000, E1   -42.273, E3 +343765.042}
SPL {X  -162.479, Y  +684.035, Z    +0.000, E1   -42.168, E3 +343777.379}
SPL {X  -162.026, Y  +689.560, Z    +0.000, E1   -42.192, E3 +343789.868}
SPL {X  -161.446, Y  +694.609, Z    +0.000, E1   -42.094, E3 +343802.000}
SPL {X  -160.889, Y  +698.503, Z    +0.000, E1   -41.849, E3 +343812.274}
SPL {X  -160.100, Y  +703.138, Z    +0.000, E1   -41.824, E3 +343823.132}
SPL {X  -158.994, Y  +708.588, Z    +0.000, E1   -41.616, E3 +343836.851}
SPL {X  -157.709, Y  +713.973, Z    +0.000, E1   -41.360, E3 +343850.634}
SPL {X  -156.530, Y  +718.319, Z    +0.000, E1   -41.164, E3 +343861.578}
SPL {X  -155.547, Y  +721.618, Z    +0.000, E1   -40.968, E3 +343870.202}
SPL {X  -151.388, Y  +733.433, Z    +0.000, E1   -44.269, E3 +343877.905}
SPL {X  -144.352, Y  +748.818, Z    +0.000, E1   -40.701, E3 +343946.940}
SPL {X  -143.859, Y  +749.757, Z    +0.000, E1   -39.148, E3 +343974.888}
ENDSPLINE

SPLINE
SPL {X  -159.245, Y  +707.432, Z    +0.000, E1   -21.244, E3 +344006.921}
SPL {X  -162.277, Y  +686.791, Z    +0.000, E1   -10.607, E3 +344008.332}
SPL {X  -162.766, Y  +677.687, Z    +0.000, E1    -5.239, E3 +344010.521}
SPL {X  -162.820, Y  +671.059, Z    +0.000, E1    -0.934, E3 +344010.877}
SPL {X  -162.820, Y  +665.599, Z    +0.000, E1    +3.424, E3 +344011.327}
SPL {X  -162.820, Y  +661.024, Z    +0.000, E1    +7.880, E3 +344010.796}
SPL {X  -162.820, Y  +654.280, Z    +0.000, E1   +14.617, E3 +344011.513}
SPL {X  -162.820, Y  +638.947, Z    +0.000, E1   +31.033, E3 +344009.566}
SPL {X  -162.820, Y  +608.150, Z    +0.000, E1   +43.921, E3 +344035.799}
SPL {X  -162.820, Y  +574.255, Z    +0.000, E1   +46.562, E3 +344085.593}
ENDSPLINE

SPLINE
SPL {X  -162.820, Y  +579.440, Z    +0.000, E1   +42.450, E3 +344098.781}
ENDSPLINE

SPLINE
SPL {X  -162.820, Y  +574.443, Z    +0.000, E1   +42.333, E3 +344110.876}
SPL {X  -162.820, Y  +568.554, Z    +0.000, E1   +42.362, E3 +344124.238}
SPL {X  -162.820, Y  +561.474, Z    +0.000, E1   +42.369, E3 +344140.423}
SPL {X  -162.820, Y  +554.421, Z    +0.000, E1   +42.414, E3 +344156.247}
SPL {X  -162.820, Y  +547.774, Z    +0.000, E1   +42.344, E3 +344171.821}
SPL {X  -162.820, Y  +541.056, Z    +0.000, E1   +42.452, E3 +344186.482}
SPL {X  -162.820, Y  +535.223, Z    +0.000, E1   +42.386, E3 +344200.176}
SPL {X  -162.820, Y  +529.084, Z    +0.000, E1   +42.400, E3 +344214.099}
SPL {X  -162.820, Y  +524.911, Z    +0.000, E1   +42.325, E3 +344223.945}
SPL {X  -162.820, Y  +519.984, Z    +0.000, E1   +42.385, E3 +344235.015}
SPL {X  -162.820, Y  +512.536, Z    +0.000, E1   +42.385, E3 +344252.126}
SPL {X  -162.820, Y  +505.746, Z    +0.000, E1   +42.400, E3 +344267.370}
SPL {X  -162.820, Y  +500.461, Z    +0.000, E1   +42.387, E3 +344279.498}
SPL {X  -162.820, Y  +494.841, Z    +0.000, E1   +42.316, E3 +344292.824}
SPL {X  -162.820, Y  +486.958, Z    +0.000, E1   +42.460, E3 +344310.117}
SPL {X  -162.820, Y  +466.305, Z    +0.000, E1   +47.564, E3 +344323.124}
SPL {X  -162.820, Y  +462.532, Z    +0.000, E1   +47.610, E3 +344330.008}
SPL {X  -162.820, Y  +458.830, Z    +0.000, E1   +46.994, E3 +344341.008}
SPL {X  -162.820, Y  +455.537, Z    +0.000, E1   +45.900, E3 +344353.827}
SPL {X  -162.820, Y  +451.000, Z    +0.000, E1   +45.084, E3 +344368.202}
SPL {X  -162.820, Y  +442.850, Z    +0.000, E1   +44.856, E3 +344386.579}
SPL {X  -162.820, Y  +435.902, Z    +0.000, E1   +44.853, E3 +344400.944}
SPL {X  -162.820, Y  +429.336, Z    +0.000, E1   +44.917, E3 +344414.462}
SPL {X  -162.820, Y  +423.193, Z    +0.000, E1   +44.819, E3 +344427.721}
SPL {X  -162.820, Y  +416.810, Z    +0.000, E1   +44.932, E3 +344440.609}
SPL {X  -162.820, Y  +408.782, Z    +0.000, E1   +44.820, E3 +344458.040}
SPL {X  -162.820, Y  +401.619, Z    +0.000, E1   +44.978, E3 +344471.961}
SPL {X  -162.820, Y  +394.771, Z    +0.000, E1   +44.856, E3 +344487.201}
SPL {X  -162.820, Y  +387.883, Z    +0.000, E1   +44.837, E3 +344501.554}
SPL {X  -162.820, Y  +382.755, Z    +0.000, E1   +44.828, E3 +344512.347}
SPL {X  -162.796, Y  +377.700, Z    +0.000, E1   +44.829, E3 +344522.928}
SPL {X  -162.619, Y  +372.412, Z    +0.000, E1   +44.928, E3 +344533.387}
SPL {X  -162.311, Y  +367.633, Z    +0.000, E1   +44.798, E3 +344544.154}
SPL {X  -161.766, Y  +362.002, Z    +0.000, E1   +44.644, E3 +344556.913}
SPL {X  -161.043, Y  +356.508, Z    +0.000, E1   +44.528, E3 +344569.027}
SPL {X  -160.417, Y  +352.631, Z    +0.000, E1   +44.411, E3 +344577.758}
SPL {X  -159.536, Y  +347.962, Z    +0.000, E1   +44.302, E3 +344588.285}
SPL {X  -158.195, Y  +341.969, Z    +0.000, E1   +44.082, E3 +344602.067}
SPL {X  -156.950, Y  +337.174, Z    +0.000, E1   +43.768, E3 +344613.758}
SPL {X  -155.654, Y  +332.729, Z    +0.000, E1   +43.534, E3 +344624.400}
SPL {X  -153.067, Y  +324.996, Z    +0.000, E1   +44.257, E3 +344636.454}
SPL {X  -147.786, Y  +312.164, Z    +0.000, E1   +47.292, E3 +344645.185}
SPL {X  -142.680, Y  +302.060, Z    +0.000, E1   +42.084, E3 +344708.557}
ENDSPLINE

SPLINE
SPL {X  -151.184, Y  +320.053, Z    +0.000, E1   +32.435, E3 +344775.800}
SPL {X  -158.917, Y  +345.064, Z    +0.000, E1   +21.858, E3 +344777.148}
SPL {X  -161.350, Y  +358.672, Z    +0.000, E1   +15.089, E3 +344779.851}
SPL {X  -162.491, Y  +370.147, Z    +0.000, E1    +8.815, E3 +344782.786}
SPL {X  -162.771, Y  +376.522, Z    +0.000, E1    +5.005, E3 +344782.395}
SPL {X  -162.820, Y  +381.116, Z    +0.000, E1    +2.017, E3 +344782.729}
SPL {X  -162.820, Y  +384.427, Z    +0.000, E1    -0.390, E3 +344783.133}
SPL {X  -162.820, Y  +387.736, Z    +0.000, E1    -3.142, E3 +344782.413}
SPL {X  -162.820, Y  +391.456, Z    +0.000, E1    -6.603, E3 +344783.200}
SPL {X  -162.820, Y  +397.032, Z    +0.000, E1   -12.435, E3 +344782.647}
SPL {X  -162.820, Y  +406.111, Z    +0.000, E1   -22.010, E3 +344783.699}
SPL {X  -162.820, Y  +418.653, Z    +0.000, E1   -36.657, E3 +344778.051}
SPL {X  -162.820, Y  +440.590, Z    +0.000, E1   -50.152, E3 +344783.297}
SPL {X  -162.820, Y  +447.889, Z    +0.000, E1   -43.424, E3 +344814.443}
SPL {X  -162.820, Y  +479.020, Z    +0.000, E1   -47.189, E3 +344854.019}
ENDSPLINE

SPLINE
SPL {X  -162.820, Y  +474.886, Z    +0.000, E1   -43.721, E3 +344865.903}
ENDSPLINE

SPLINE
SPL {X  -162.820, Y  +476.137, Z    +0.000, E1   -42.304, E3 +344877.017}
SPL {X  -162.820, Y  +480.895, Z    +0.000, E1   -42.223, E3 +344888.476}
SPL {X  -162.820, Y  +485.782, Z    +0.000, E1   -42.348, E3 +344898.821}
SPL {X  -162.820, Y  +489.480, Z    +0.000, E1   -42.230, E3 +344908.048}
SPL {X  -162.820, Y  +494.825, Z    +0.000, E1   -42.287, E3 +344919.996}
SPL {X  -162.820, Y  +501.909, Z    +0.000, E1   -42.324, E3 +344936.182}
SPL {X  -162.820, Y  +508.157, Z    +0.000, E1   -42.280, E3 +344950.513}
SPL {X  -162.820, Y  +513.215, Z    +0.000, E1   -42.304, E3 +344962.043}
SPL {X  -162.820, Y  +520.311, Z    +0.000, E1   -42.317, E3 +344978.341}
SPL {X  -162.820, Y  +526.529, Z    +0.000, E1   -42.247, E3 +344992.811}
SPL {X  -162.820, Y  +531.715, Z    +0.000, E1   -42.312, E3 +345004.333}
SPL {X  -162.820, Y  +537.459, Z    +0.000, E1   -42.308, E3 +345017.592}
SPL {X  -162.820, Y  +542.643, Z    +0.000, E1   -42.173, E3 +345030.184}
SPL {X  -162.820, Y  +549.160, Z    +0.000, E1   -42.387, E3 +345043.943}
SPL {X  -162.820, Y  +554.884, Z    +0.000, E1   -42.207, E3 +345058.028}
SPL {X  -162.820, Y  +561.114, Z    +0.000, E1   -42.336, E3 +345071.608}
SPL {X  -162.820, Y  +566.097, Z    +0.000, E1   -42.118, E3 +345084.219}
SPL {X  -162.820, Y  +571.654, Z    +0.000, E1   -42.313, E3 +345095.872}
SPL {X  -162.820, Y  +577.246, Z    +0.000, E1   -42.284, E3 +345108.837}
SPL {X  -162.820, Y  +582.233, Z    +0.000, E1   -42.188, E3 +345120.817}
SPL {X  -162.820, Y  +588.138, Z    +0.000, E1   -42.308, E3 +345133.715}
SPL {X  -162.820, Y  +593.999, Z    +0.000, E1   -42.301, E3 +345147.125}
SPL {X  -162.820, Y  +599.194, Z    +0.000, E1   -42.235, E3 +345159.430}
SPL {X  -162.820, Y  +604.595, Z    +0.000, E1   -42.290, E3 +345171.461}
SPL {X  -162.820, Y  +609.630, Z    +0.000, E1   -42.276, E3 +345183.087}
SPL {X  -162.820, Y  +614.392, Z    +0.000, E1   -42.242, E3 +345194.187}
SPL {X  -162.820, Y  +620.424, Z    +0.000, E1   -42.277, E3 +345207.935}
SPL {X  -162.820, Y  +626.430, Z    +0.000, E1   -42.291, E3 +345221.485}
SPL {X  -162.820, Y  +631.865, Z    +0.000, E1   -42.327, E3 +345233.778}
SPL {X  -162.820, Y  +637.189, Z    +0.000, E1   -42.236, E3 +345246.452}
SPL {X  -162.820, Y  +642.066, Z    +0.000, E1   -42.247, E3 +345257.574}
SPL {X  -162.820, Y  +646.907, Z    +0.000, E1   -42.249, E3 +345268.693}
SPL {X  -162.820, Y  +652.374, Z    +0.000, E1   -42.262, E3 +345281.132}
SPL {X  -162.820, Y  +657.439, Z    +0.000, E1   -42.251, E3 +345292.805}
SPL {X  -162.820, Y  +663.328, Z    +0.000, E1   -42.283, E3 +345306.207}
SPL {X  -162.820, Y  +669.078, Z    +0.000, E1   -42.263, E3 +345319.403}
SPL {X  -162.819, Y  +673.910, Z    +0.000, E1   -42.244, E3 +345330.597}
SPL {X  -162.729, Y  +678.944, Z    +0.000, E1   -42.273, E3 +345341.965}
SPL {X  -162.479, Y  +684.035, Z    +0.000, E1   -42.168, E3 +345354.302}
SPL {X  -162.026, Y  +689.560, Z    +0.000, E1   -42.192, E3 +345366.791}
SPL {X  -161.446, Y  +694.609, Z    +0.000, E1   -42.094, E3 +345378.923}
SPL {X  -160.681, Y  +699.806, Z    +0.000, E1   -41.866, E3 +345392.206}
SPL {X  -159.658, Y  +705.434, Z    +0.000, E1   -41.735, E3 +345405.836}
SPL {X  -158.502, Y  +710.748, Z    +0.000, E1   -41.532, E3 +345419.183}
SPL {X  -157.452, Y  +714.962, Z    +0.000, E1   -41.276, E3 +345430.178}
SPL {X  -156.530, Y  +718.319, Z    +0.000, E1   -41.164, E3 +345438.501}
SPL {X  -155.547, Y  +721.618, Z    +0.000, E1   -40.968, E3 +345447.125}
SPL {X  -151.388, Y  +733.433, Z    +0.000, E1   -44.269, E3 +345454.828}
SPL {X  -144.352, Y  +748.818, Z    +0.000, E1   -40.701, E3 +345523.863}
SPL {X  -143.859, Y  +749.757, Z    +0.000, E1   -39.148, E3 +345551.811}
ENDSPLINE

SPLINE
SPL {X  -159.245, Y  +707.432, Z    +0.000, E1   -21.244, E3 +345583.844}
SPL {X  -162.277, Y  +686.791, Z    +0.000, E1   -10.607, E3 +345585.255}
SPL {X  -162.766, Y  +677.687, Z    +0.000, E1    -5.239, E3 +345587.444}
SPL {X  -162.820, Y  +671.059, Z    +0.000, E1    -0.934, E3 +345587.800}
SPL {X  -162.820, Y  +665.599, Z    +0.000, E1    +3.424, E3 +345588.250}
SPL {X  -162.820, Y  +661.024, Z    +0.000, E1    +7.880, E3 +345587.719}
SPL {X  -162.820, Y  +656.051, Z    +0.000, E1   +12.848, E3 +345588.586}
SPL {X  -162.820, Y  +650.794, Z    +0.000, E1   +18.580, E3 +345588.142}
SPL {X  -162.820, Y  +638.947, Z    +0.000, E1   +31.033, E3 +345586.490}
SPL {X  -162.820, Y  +608.150, Z    +0.000, E1   +43.921, E3 +345612.722}
SPL {X  -162.820, Y  +574.255, Z    +0.000, E1   +46.562, E3 +345662.516}
ENDSPLINE

SPLINE
SPL {X  -162.820, Y  +579.440, Z    +0.000, E1   +42.450, E3 +345675.704}
ENDSPLINE

SPLINE
SPL {X  -162.820, Y  +574.443, Z    +0.000, E1   +42.333, E3 +345687.799}
SPL {X  -162.820, Y  +568.554, Z    +0.000, E1   +42.362, E3 +345701.161}
SPL {X  -162.820, Y  +561.474, Z    +0.000, E1   +42.369, E3 +345717.346}
SPL {X  -162.820, Y  +555.861, Z    +0.000, E1   +42.349, E3 +345730.151}
SPL {X  -162.820, Y  +550.633, Z    +0.000, E1   +42.421, E3 +345741.681}
SPL {X  -162.820, Y  +546.534, Z    +0.000, E1   +42.268, E3 +345751.890}
SPL {X  -162.820, Y  +539.632, Z    +0.000, E1   +42.488, E3 +345766.611}
SPL {X  -162.820, Y  +533.959, Z    +0.000, E1   +42.310, E3 +345780.308}
SPL {X  -162.820, Y  +527.661, Z    +0.000, E1   +42.425, E3 +345794.304}
SPL {X  -162.820, Y  +521.246, Z    +0.000, E1   +42.365, E3 +345809.057}
SPL {X  -162.820, Y  +515.708, Z    +0.000, E1   +42.333, E3 +345822.019}
SPL {X  -162.820, Y  +510.265, Z    +0.000, E1   +42.390, E3 +345833.981}
SPL {X  -162.820, Y  +505.746, Z    +0.000, E1   +42.400, E3 +345844.293}
SPL {X  -162.820, Y  +500.461, Z    +0.000, E1   +42.387, E3 +345856.421}
SPL {X  -162.820, Y  +494.841, Z    +0.000, E1   +42.316, E3 +345869.747}
SPL {X  -162.820, Y  +486.958, Z    +0.000, E1   +42.460, E3 +345887.040}
SPL {X  -162.820, Y  +464.528, Z    +0.000, E1   +47.611, E3 +345903.253}
SPL {X  -162.820, Y  +458.830, Z    +0.000, E1   +46.994, E3 +345917.931}
SPL {X  -162.820, Y  +455.537, Z    +0.000, E1   +45.900, E3 +345930.750}
SPL {X  -162.820, Y  +452.032, Z    +0.000, E1   +45.224, E3 +345941.955}
SPL {X  -162.820, Y  +446.617, Z    +0.000, E1   +44.768, E3 +345956.041}
SPL {X  -162.820, Y  +440.464, Z    +0.000, E1   +44.845, E3 +345968.343}
SPL {X  -162.820, Y  +435.902, Z    +0.000, E1   +44.853, E3 +345977.867}
SPL {X  -162.820, Y  +429.336, Z    +0.000, E1   +44.917, E3 +345991.385}
SPL {X  -162.820, Y  +423.193, Z    +0.000, E1   +44.819, E3 +346004.644}
SPL {X  -162.820, Y  +416.810, Z    +0.000, E1   +44.932, E3 +346017.532}
SPL {X  -162.820, Y  +408.782, Z    +0.000, E1   +44.820, E3 +346034.963}
SPL {X  -162.820, Y  +401.619, Z    +0.000, E1   +44.978, E3 +346048.885}
SPL {X  -162.820, Y  +394.771, Z    +0.000, E1   +44.856, E3 +346064.124}
SPL {X  -162.820, Y  +387.883, Z    +0.000, E1   +44.837, E3 +346078.478}
SPL {X  -162.820, Y  +382.755, Z    +0.000, E1   +44.828, E3 +346089.271}
SPL {X  -162.796, Y  +377.700, Z    +0.000, E1   +44.829, E3 +346099.851}
SPL {X  -162.619, Y  +372.412, Z    +0.000, E1   +44.928, E3 +346110.310}
SPL {X  -162.311, Y  +367.633, Z    +0.000, E1   +44.798, E3 +346121.077}
SPL {X  -161.766, Y  +362.002, Z    +0.000, E1   +44.644, E3 +346133.836}
SPL {X  -161.043, Y  +356.508, Z    +0.000, E1   +44.528, E3 +346145.950}
SPL {X  -160.070, Y  +350.699, Z    +0.000, E1   +44.409, E3 +346158.902}
SPL {X  -158.853, Y  +344.776, Z    +0.000, E1   +44.148, E3 +346172.723}
SPL {X  -157.292, Y  +338.433, Z    +0.000, E1   +43.917, E3 +346187.401}
SPL {X  -155.654, Y  +332.729, Z    +0.000, E1   +43.534, E3 +346201.323}
SPL {X  -154.189, Y  +328.191, Z    +0.000, E1   +43.338, E3 +346211.820}
SPL {X  -149.333, Y  +315.614, Z    +0.000, E1   +46.650, E3 +346219.135}
SPL {X  -142.680, Y  +302.060, Z    +0.000, E1   +42.084, E3 +346285.480}
ENDSPLINE

SPLINE
SPL {X  -151.184, Y  +320.053, Z    +0.000, E1   +32.435, E3 +346352.723}
SPL {X  -158.917, Y  +345.064, Z    +0.000, E1   +21.858, E3 +346354.071}
SPL {X  -161.350, Y  +358.672, Z    +0.000, E1   +15.089, E3 +346356.774}
SPL {X  -162.491, Y  +370.147, Z    +0.000, E1    +8.815, E3 +346359.709}
SPL {X  -162.816, Y  +379.394, Z    +0.000, E1    +3.267, E3 +346359.536}
SPL {X  -162.820, Y  +384.427, Z    +0.000, E1    -0.390, E3 +346360.056}
SPL {X  -162.820, Y  +387.736, Z    +0.000, E1    -3.142, E3 +346359.337}
SPL {X  -162.820, Y  +391.456, Z    +0.000, E1    -6.603, E3 +346360.123}
SPL {X  -162.820, Y  +397.032, Z    +0.000, E1   -12.435, E3 +346359.570}
SPL {X  -162.820, Y  +406.111, Z    +0.000, E1   -22.010, E3 +346360.622}
SPL {X  -162.820, Y  +418.653, Z    +0.000, E1   -36.657, E3 +346354.974}
SPL {X  -162.820, Y  +440.590, Z    +0.000, E1   -50.152, E3 +346360.220}
SPL {X  -162.820, Y  +447.889, Z    +0.000, E1   -43.424, E3 +346391.366}
SPL {X  -162.820, Y  +478.087, Z    +0.000, E1   -45.903, E3 +346436.585}
ENDSPLINE

SPLINE
SPL {X  -162.820, Y  +474.900, Z    +0.000, E1   -42.394, E3 +346450.737}
ENDSPLINE

SPLINE
SPL {X  -162.820, Y  +480.895, Z    +0.000, E1   -42.223, E3 +346465.399}
SPL {X  -162.820, Y  +485.782, Z    +0.000, E1   -42.348, E3 +346475.744}
SPL {X  -162.820, Y  +489.480, Z    +0.000, E1   -42.230, E3 +346484.971}
SPL {X  -162.820, Y  +494.825, Z    +0.000, E1   -42.287, E3 +346496.919}
SPL {X  -162.820, Y  +501.023, Z    +0.000, E1   -42.347, E3 +346510.801}
SPL {X  -162.820, Y  +506.968, Z    +0.000, E1   -42.248, E3 +346524.992}
SPL {X  -162.820, Y  +513.215, Z    +0.000, E1   -42.304, E3 +346538.966}
SPL {X  -162.820, Y  +518.708, Z    +0.000, E1   -42.272, E3 +346551.688}
SPL {X  -162.820, Y  +525.147, Z    +0.000, E1   -42.298, E3 +346566.430}
SPL {X  -162.820, Y  +531.715, Z    +0.000, E1   -42.312, E3 +346581.256}
SPL {X  -162.820, Y  +537.459, Z    +0.000, E1   -42.308, E3 +346594.515}
SPL {X  -162.820, Y  +542.643, Z    +0.000, E1   -42.173, E3 +346607.107}
SPL {X  -162.820, Y  +549.160, Z    +0.000, E1   -42.387, E3 +346620.866}
SPL {X  -162.820, Y  +554.884, Z    +0.000, E1   -42.207, E3 +346634.951}
SPL {X  -162.820, Y  +561.114, Z    +0.000, E1   -42.336, E3 +346648.531}
SPL {X  -162.820, Y  +566.097, Z    +0.000, E1   -42.118, E3 +346661.142}
SPL {X  -162.820, Y  +571.654, Z    +0.000, E1   -42.313, E3 +346672.795}
SPL {X  -162.820, Y  +577.246, Z    +0.000, E1   -42.284, E3 +346685.760}
SPL {X  -162.820, Y  +582.233, Z    +0.000, E1   -42.188, E3 +346697.740}
SPL {X  -162.820, Y  +588.138, Z    +0.000, E1   -42.308, E3 +346710.638}
SPL {X  -162.820, Y  +593.999, Z    +0.000, E1   -42.301, E3 +346724.048}
SPL {X  -162.820, Y  +599.194, Z    +0.000, E1   -42.235, E3 +346736.353}
SPL {X  -162.820, Y  +604.595, Z    +0.000, E1   -42.290, E3 +346748.384}
SPL {X  -162.820, Y  +609.630, Z    +0.000, E1   -42.276, E3 +346760.010}
SPL {X  -162.820, Y  +614.392, Z    +0.000, E1   -42.242, E3 +346771.110}
SPL {X  -162.820, Y  +620.424, Z    +0.000, E1   -42.277, E3 +346784.858}
SPL {X  -162.820, Y  +626.430, Z    +0.000, E1   -42.291, E3 +346798.408}
SPL {X  -162.820, Y  +631.865, Z    +0.000, E1   -42.327, E3 +346810.701}
SPL {X  -162.820, Y  +637.189, Z    +0.000, E1   -42.236, E3 +346823.375}
SPL {X  -162.820, Y  +642.066, Z    +0.000, E1   -42.247, E3 +346834.497}
SPL {X  -162.820, Y  +646.907, Z    +0.000, E1   -42.249, E3 +346845.617}
SPL {X  -162.820, Y  +652.374, Z    +0.000, E1   -42.262, E3 +346858.055}
SPL {X  -162.820, Y  +657.439, Z    +0.000, E1   -42.251, E3 +346869.728}
SPL {X  -162.820, Y  +663.328, Z    +0.000, E1   -42.283, E3 +346883.130}
SPL {X  -162.820, Y  +669.078, Z    +0.000, E1   -42.263, E3 +346896.326}
SPL {X  -162.819, Y  +673.910, Z    +0.000, E1   -42.244, E3 +346907.520}
SPL {X  -162.729, Y  +678.944, Z    +0.000, E1   -42.273, E3 +346918.888}
SPL {X  -162.479, Y  +684.035, Z    +0.000, E1   -42.168, E3 +346931.225}
SPL {X  -162.026, Y  +689.560, Z    +0.000, E1   -42.192, E3 +346943.714}
SPL {X  -161.446, Y  +694.609, Z    +0.000, E1   -42.094, E3 +346955.846}
SPL {X  -160.889, Y  +698.503, Z    +0.000, E1   -41.849, E3 +346966.120}
SPL {X  -160.100, Y  +703.138, Z    +0.000, E1   -41.824, E3 +346976.978}
SPL {X  -158.994, Y  +708.588, Z    +0.000, E1   -41.616, E3 +346990.698}
SPL {X  -157.709, Y  +713.973, Z    +0.000, E1   -41.360, E3 +347004.480}
SPL {X  -156.530, Y  +718.319, Z    +0.000, E1   -41.164, E3 +347015.424}
SPL {X  -155.547, Y  +721.618, Z    +0.000, E1   -40.968, E3 +347024.048}
SPL {X  -151.388, Y  +733.433, Z    +0.000, E1   -44.269, E3 +347031.751}
SPL {X  -144.352, Y  +748.818, Z    +0.000, E1   -40.701, E3 +347100.786}
SPL {X  -143.859, Y  +749.757, Z    +0.000, E1   -39.148, E3 +347128.734}
ENDSPLINE

SPLINE
SPL {X  -159.245, Y  +707.432, Z    +0.000, E1   -21.244, E3 +347160.767}
SPL {X  -162.277, Y  +686.791, Z    +0.000, E1   -10.607, E3 +347162.178}
SPL {X  -162.766, Y  +677.687, Z    +0.000, E1    -5.239, E3 +347164.368}
SPL {X  -162.820, Y  +671.059, Z    +0.000, E1    -0.934, E3 +347164.724}
SPL {X  -162.820, Y  +665.599, Z    +0.000, E1    +3.424, E3 +347165.173}
SPL {X  -162.820, Y  +661.024, Z    +0.000, E1    +7.880, E3 +347164.642}
SPL {X  -162.820, Y  +654.280, Z    +0.000, E1   +14.617, E3 +347165.359}
SPL {X  -162.820, Y  +638.947, Z    +0.000, E1   +31.033, E3 +347163.413}
SPL {X  -162.820, Y  +608.150, Z    +0.000, E1   +43.921, E3 +347189.645}
SPL {X  -162.820, Y  +574.255, Z    +0.000, E1   +46.562, E3 +347239.439}
ENDSPLINE

SPLINE
SPL {X  -162.820, Y  +579.440, Z    +0.000, E1   +42.450, E3 +347252.627}
ENDSPLINE

SPLINE
SPL {X  -162.820, Y  +574.443, Z    +0.000, E1   +42.333, E3 +347264.722}
SPL {X  -162.820, Y  +568.554, Z    +0.000, E1   +42.362, E3 +347278.084}
SPL {X  -162.820, Y  +561.474, Z    +0.000, E1   +42.369, E3 +347294.269}
SPL {X  -162.820, Y  +555.861, Z    +0.000, E1   +42.349, E3 +347307.074}
SPL {X  -162.820, Y  +550.633, Z    +0.000, E1   +42.421, E3 +347318.604}
SPL {X  -162.820, Y  +546.534, Z    +0.000, E1   +42.268, E3 +347328.813}
SPL {X  -162.820, Y  +541.056, Z    +0.000, E1   +42.452, E3 +347340.328}
SPL {X  -162.820, Y  +535.223, Z    +0.000, E1   +42.386, E3 +347354.022}
SPL {X  -162.820, Y  +529.084, Z    +0.000, E1   +42.400, E3 +347367.945}
SPL {X  -162.820, Y  +522.568, Z    +0.000, E1   +42.385, E3 +347382.975}
SPL {X  -162.820, Y  +515.708, Z    +0.000, E1   +42.333, E3 +347398.942}
SPL {X  -162.820, Y  +510.265, Z    +0.000, E1   +42.390, E3 +347410.904}
SPL {X  -162.820, Y  +505.746, Z    +0.000, E1   +42.400, E3 +347421.216}
SPL {X  -162.820, Y  +500.461, Z    +0.000, E1   +42.387, E3 +347433.344}
SPL {X  -162.820, Y  +494.841, Z    +0.000, E1   +42.316, E3 +347446.670}
SPL {X  -162.820, Y  +487.903, Z    +0.000, E1   +42.488, E3 +347461.493}
SPL {X  -162.820, Y  +484.250, Z    +0.000, E1   +42.201, E3 +347471.354}
SPL {X  -162.820, Y  +464.528, Z    +0.000, E1   +47.611, E3 +347480.176}
SPL {X  -162.820, Y  +459.899, Z    +0.000, E1   +47.097, E3 +347492.019}
SPL {X  -162.820, Y  +455.990, Z    +0.000, E1   +46.212, E3 +347505.093}
SPL {X  -162.820, Y  +452.032, Z    +0.000, E1   +45.224, E3 +347518.878}
SPL {X  -162.820, Y  +446.617, Z    +0.000, E1   +44.768, E3 +347532.965}
SPL {X  -162.820, Y  +437.902, Z    +0.000, E1   +44.900, E3 +347550.541}
SPL {X  -162.820, Y  +430.894, Z    +0.000, E1   +44.976, E3 +347564.527}
SPL {X  -162.820, Y  +425.053, Z    +0.000, E1   +44.824, E3 +347577.789}
SPL {X  -162.820, Y  +418.403, Z    +0.000, E1   +44.941, E3 +347590.902}
SPL {X  -162.820, Y  +412.479, Z    +0.000, E1   +44.780, E3 +347604.332}
SPL {X  -162.820, Y  +406.707, Z    +0.000, E1   +44.849, E3 +347615.905}
SPL {X  -162.820, Y  +400.166, Z    +0.000, E1   +44.948, E3 +347629.189}
SPL {X  -162.820, Y  +393.279, Z    +0.000, E1   +44.825, E3 +347644.192}
SPL {X  -162.820, Y  +387.883, Z    +0.000, E1   +44.837, E3 +347655.401}
SPL {X  -162.820, Y  +382.755, Z    +0.000, E1   +44.828, E3 +347666.194}
SPL {X  -162.796, Y  +377.700, Z    +0.000, E1   +44.829, E3 +347676.774}
SPL {X  -162.619, Y  +372.412, Z    +0.000, E1   +44.928, E3 +347687.233}
SPL {X  -162.170, Y  +365.961, Z    +0.000, E1   +44.802, E3 +347701.663}
SPL {X  -161.259, Y  +358.011, Z    +0.000, E1   +44.581, E3 +347719.590}
SPL {X  -160.417, Y  +352.631, Z    +0.000, E1   +44.411, E3 +347731.605}
SPL {X  -159.784, Y  +349.204, Z    +0.000, E1   +44.340, E3 +347739.197}
SPL {X  -158.853, Y  +344.776, Z    +0.000, E1   +44.148, E3 +347749.646}
SPL {X  -157.292, Y  +338.433, Z    +0.000, E1   +43.917, E3 +347764.324}
SPL {X  -155.654, Y  +332.729, Z    +0.000, E1   +43.534, E3 +347778.246}
SPL {X  -154.189, Y  +328.191, Z    +0.000, E1   +43.338, E3 +347788.743}
SPL {X  -149.333, Y  +315.614, Z    +0.000, E1   +46.650, E3 +347796.059}
SPL {X  -142.680, Y  +302.060, Z    +0.000, E1   +42.084, E3 +347862.403}
ENDSPLINE

SPLINE
SPL {X  -151.184, Y  +320.053, Z    +0.000, E1   +32.435, E3 +347929.646}
SPL {X  -158.917, Y  +345.064, Z    +0.000, E1   +21.858, E3 +347930.994}
SPL {X  -161.350, Y  +358.672, Z    +0.000, E1   +15.089, E3 +347933.697}
SPL {X  -162.491, Y  +370.147, Z    +0.000, E1    +8.815, E3 +347936.632}
SPL {X  -162.816, Y  +379.394, Z    +0.000, E1    +3.267, E3 +347936.459}
SPL {X  -162.820, Y  +384.427, Z    +0.000, E1    -0.390, E3 +347936.979}
SPL {X  -162.820, Y  +387.736, Z    +0.000, E1    -3.142, E3 +347936.260}
SPL {X  -162.820, Y  +391.456, Z    +0.000, E1    -6.603, E3 +347937.046}
SPL {X  -162.820, Y  +397.032, Z    +0.000, E1   -12.435, E3 +347936.493}
SPL {X  -162.820, Y  +406.111, Z    +0.000, E1   -22.010, E3 +347937.545}
SPL {X  -162.820, Y  +418.653, Z    +0.000, E1   -36.657, E3 +347931.897}
SPL {X  -162.820, Y  +440.590, Z    +0.000, E1   -50.152, E3 +347937.143}
SPL {X  -162.820, Y  +447.889, Z    +0.000, E1   -43.424, E3 +347968.289}
SPL {X  -162.820, Y  +478.087, Z    +0.000, E1   -45.903, E3 +348013.508}
ENDSPLINE

SPLINE
SPL {X  -162.820, Y  +472.818, Z    +0.000, E1   -42.437, E3 +348022.449}
ENDSPLINE

SPLINE
SPL {X  -162.820, Y  +476.137, Z    +0.000, E1   -42.304, E3 +348030.863}
SPL {X  -162.820, Y  +480.895, Z    +0.000, E1   -42.223, E3 +348042.322}
SPL {X  -162.820, Y  +488.112, Z    +0.000, E1   -42.323, E3 +348058.403}
SPL {X  -162.820, Y  +496.300, Z    +0.000, E1   -42.332, E3 +348077.115}
SPL {X  -162.820, Y  +503.162, Z    +0.000, E1   -42.272, E3 +348093.032}
SPL {X  -162.820, Y  +508.157, Z    +0.000, E1   -42.280, E3 +348104.359}
SPL {X  -162.820, Y  +513.215, Z    +0.000, E1   -42.304, E3 +348115.889}
SPL {X  -162.820, Y  +520.311, Z    +0.000, E1   -42.317, E3 +348132.188}
SPL {X  -162.820, Y  +526.529, Z    +0.000, E1   -42.247, E3 +348146.657}
SPL {X  -162.820, Y  +532.723, Z    +0.000, E1   -42.344, E3 +348160.399}
SPL {X  -162.820, Y  +538.500, Z    +0.000, E1   -42.256, E3 +348174.020}
SPL {X  -162.820, Y  +542.643, Z    +0.000, E1   -42.173, E3 +348184.030}
SPL {X  -162.820, Y  +549.160, Z    +0.000, E1   -42.387, E3 +348197.789}
SPL {X  -162.820, Y  +554.884, Z    +0.000, E1   -42.207, E3 +348211.874}
SPL {X  -162.820, Y  +559.897, Z    +0.000, E1   -42.319, E3 +348222.660}
SPL {X  -162.820, Y  +565.154, Z    +0.000, E1   -42.205, E3 +348235.506}
SPL {X  -162.820, Y  +571.654, Z    +0.000, E1   -42.313, E3 +348249.718}
SPL {X  -162.820, Y  +577.246, Z    +0.000, E1   -42.284, E3 +348262.684}
SPL {X  -162.820, Y  +582.233, Z    +0.000, E1   -42.188, E3 +348274.663}
SPL {X  -162.820, Y  +588.138, Z    +0.000, E1   -42.308, E3 +348287.561}
SPL {X  -162.820, Y  +593.999, Z    +0.000, E1   -42.301, E3 +348300.971}
SPL {X  -162.820, Y  +599.194, Z    +0.000, E1   -42.235, E3 +348313.276}
SPL {X  -162.820, Y  +604.595, Z    +0.000, E1   -42.290, E3 +348325.307}
SPL {X  -162.820, Y  +609.630, Z    +0.000, E1   -42.276, E3 +348336.933}
SPL {X  -162.820, Y  +614.392, Z    +0.000, E1   -42.242, E3 +348348.033}
SPL {X  -162.820, Y  +620.424, Z    +0.000, E1   -42.277, E3 +348361.781}
SPL {X  -162.820, Y  +626.430, Z    +0.000, E1   -42.291, E3 +348375.331}
SPL {X  -162.820, Y  +631.865, Z    +0.000, E1   -42.327, E3 +348387.624}
SPL {X  -162.820, Y  +637.189, Z    +0.000, E1   -42.236, E3 +348400.298}
SPL {X  -162.820, Y  +642.066, Z    +0.000, E1   -42.247, E3 +348411.421}
SPL {X  -162.820, Y  +646.907, Z    +0.000, E1   -42.249, E3 +348422.540}
SPL {X  -162.820, Y  +652.374, Z    +0.000, E1   -42.262, E3 +348434.978}
SPL {X  -162.820, Y  +658.634, Z    +0.000, E1   -42.281, E3 +348449.335}
SPL {X  -162.820, Y  +664.480, Z    +0.000, E1   -42.257, E3 +348462.730}
SPL {X  -162.820, Y  +669.078, Z    +0.000, E1   -42.263, E3 +348473.249}
SPL {X  -162.819, Y  +673.910, Z    +0.000, E1   -42.244, E3 +348484.443}
SPL {X  -162.729, Y  +678.944, Z    +0.000, E1   -42.273, E3 +348495.811}
SPL {X  -162.479, Y  +684.035, Z    +0.000, E1   -42.168, E3 +348508.148}
SPL {X  -162.026, Y  +689.560, Z    +0.000, E1   -42.192, E3 +348520.637}
SPL {X  -161.446, Y  +694.609, Z    +0.000, E1   -42.094, E3 +348532.769}
SPL {X  -160.889, Y  +698.503, Z    +0.000, E1   -41.849, E3 +348543.043}
SPL {X  -160.100, Y  +703.138, Z    +0.000, E1   -41.824, E3 +348553.901}
SPL {X  -159.403, Y  +706.682, Z    +0.000, E1   -41.618, E3 +348563.080}
SPL {X  -158.502, Y  +710.748, Z    +0.000, E1   -41.532, E3 +348573.029}
SPL {X  -157.452, Y  +714.962, Z    +0.000, E1   -41.276, E3 +348584.025}
SPL {X  -156.258, Y  +719.258, Z    +0.000, E1   -41.133, E3 +348594.769}
SPL {X  -155.356, Y  +722.233, Z    +0.000, E1   -40.927, E3 +348602.559}
SPL {X  -151.388, Y  +733.433, Z    +0.000, E1   -44.269, E3 +348608.674}
SPL {X  -144.352, Y  +748.818, Z    +0.000, E1   -40.701, E3 +348677.709}
SPL {X  -143.859, Y  +749.757, Z    +0.000, E1   -39.148, E3 +348705.657}
ENDSPLINE

